   IF #Signal_AI.Value < #Signal_AI.Scal_Min_Eu THEN      //Ïðè âûõîäå çíà÷åíèÿ ñèãíàëà èç çàäàííîãî äèàïàçîíà ïðèðàâíèâàåì åãî ê íèæíåìó ïðåäåëó  ýòîãî äèàïàçîíà
       #Signal_AI.Value := #Signal_AI.Scal_Min_Eu;
       #Signal_AI.Scal_Min_Under := true;                 //çàæèãàåì ôëàã  çíà÷åíèÿ ñèãíàëà íèæå íèæíåãî ïðåäåëà äèàïàçîíà ìàñøòàáèðîâàíèÿ
   ELSE
       #Signal_AI.Scal_Min_Under := false;
   END_IF;

   //------------------------------------------------------------------------
   //---------Áëîê ïðîâåðêè ïðåâûøåíèÿ óñòàâêè ïî âåðõíåìó àâàðèéíîìó ïðåäåëó
   //------------------------------------------------------------------------
   IF #Signal_AI.HH_Alarm THEN    // Åñëè åñòü àâàðèÿ òî äëÿ îáåñïå÷åíèÿ ãèñòåðåçèñà 
       // Ðàçðåøåíèå íà ñòàðò òàéìåðà åñëè ïðîâåðêà ðàçðåøåíà è çíà÷åíèå ïðåâûøàåò óñòàâêó
       #Temp_Start_Timer := #Signal_AI.HH_Alarm_En AND (#Signal_AI.Value > (#Signal_AI.HH_Lim - #Signal_AI.HH_DeadBand));
   ELSE
       // Ðàçðåøåíèå íà ñòàðò òàéìåðà åñëè ïðîâåðêà ðàçðåøåíà è çíà÷åíèå ïðåâûøàåò óñòàâêó
       #Temp_Start_Timer := #Signal_AI.HH_Alarm_En AND (#Signal_AI.Value > (#Signal_AI.HH_Lim + #Signal_AI.HH_DeadBand));
   END_IF;

   #HH_Timer(IN := #Temp_Start_Timer // IN: BOOL
             ,
             PT := #Signal_AI.HH_Delay // IN: TIME
   );

   //åñëè  âðåìÿ çàäåðæêè èñòåêëî òî çàæèãàåì ôëàã àâàðèè , èíà÷å ãàñèì åãî
   IF #HH_Timer.Q THEN
       #Signal_AI.HH_Alarm := true;
       #Signal_AI.State := #Signal_AI.State OR #UEL;
   ELSE
       #Signal_AI.HH_Alarm := false;
       #Signal_AI.State := #Signal_AI.State AND (NOT (#UEL));
   END_IF;

   //------------------------------------------------------------------------
   //Áëîê ïðîâåðêè ïðåâûøåíèÿ óñòàâêè ïî âåðõíåìó ïðåäóïðåäèòåëüíîìó ïðåäåëó
   //------------------------------------------------------------------------
   IF #Signal_AI.H_Alarm THEN    // Åñëè åñòü àâàðèÿ òî äëÿ îáåñïå÷åíèÿ ãèñòåðåçèñà 
       // Ðàçðåøåíèå íà ñòàðò òàéìåðà åñëè ïðîâåðêà ðàçðåøåíà è çíà÷åíèå ïðåâûøàåò óñòàâêó
       #Temp_Start_Timer := #Signal_AI.H_Alarm_En AND (#Signal_AI.Value > (#Signal_AI.H_Lim - #Signal_AI.H_DeadBand));
   ELSE
       // Ðàçðåøåíèå íà ñòàðò òàéìåðà åñëè ïðîâåðêà ðàçðåøåíà è çíà÷åíèå ïðåâûøàåò óñòàâêó
       #Temp_Start_Timer := #Signal_AI.H_Alarm_En AND (#Signal_AI.Value > (#Signal_AI.H_Lim + #Signal_AI.H_DeadBand));
   END_IF;

   #H_Timer(IN := #Temp_Start_Timer // IN: BOOL
            ,
            PT := #Signal_AI.H_Delay // IN: TIME
   );

   //åñëè  âðåìÿ çàäåðæêè èñòåêëî òî çàæèãàåì ôëàã àâàðèè , èíà÷å ãàñèì åãî
   IF #H_Timer.Q THEN
       #Signal_AI.H_Alarm := true;
       #Signal_AI.State := #Signal_AI.State OR #UWL;
   ELSE
       #Signal_AI.H_Alarm := false;
       #Signal_AI.State := #Signal_AI.State AND (NOT (#UWL));
   END_IF;

   //------------------------------------------------------------------------
   //--Áëîê ïðîâåðêè ïðåâûøåíèÿ óñòàâêè ïî íèæíåìó ïðåäóïðåäèòåëüíîìó ïðåäåëó
   //------------------------------------------------------------------------
   IF #Signal_AI.L_Alarm THEN    // Åñëè åñòü àâàðèÿ òî äëÿ îáåñïå÷åíèÿ ãèñòåðåçèñà 
       #Temp_Start_Timer := #Signal_AI.L_Alarm_En AND (#Signal_AI.Value < (#Signal_AI.L_Lim + #Signal_AI.L_DeadBand));   // Ðàçðåøåíèå íà ñòàðò òàéìåðà åñëè ïðîâåðêà ðàçðåøåíà è çíà÷åíèå ïðåâûøàåò óñòàâêó
   ELSE
       #Temp_Start_Timer := #Signal_AI.L_Alarm_En AND (#Signal_AI.Value < (#Signal_AI.L_Lim - #Signal_AI.L_DeadBand));   // Ðàçðåøåíèå íà ñòàðò òàéìåðà åñëè ïðîâåðêà ðàçðåøåíà è çíà÷åíèå ïðåâûøàåò óñòàâêó
   END_IF;

   #L_Timer(IN := #Temp_Start_Timer // IN: BOOL
            ,
            PT := #Signal_AI.L_Delay // IN: TIME
   );

   //åñëè  âðåìÿ çàäåðæêè èñòåêëî òî çàæèãàåì ôëàã àâàðèè , èíà÷å ãàñèì åãî
   IF #L_Timer.Q THEN
       #Signal_AI.L_Alarm := true;
       #Signal_AI.State := #Signal_AI.State OR #DWL;
   ELSE
       #Signal_AI.L_Alarm := false;
       #Signal_AI.State := #Signal_AI.State AND (NOT (#DWL));
   END_IF;

   //------------------------------------------------------------------------
   //-------Áëîê ïðîâåðêè ïðåâûøåíèÿ óñòàâêè ïî íèæíåìó àâàðèéíîìó ïðåäåëó---
   //------------------------------------------------------------------------
   IF #Signal_AI.LL_Alarm THEN    // Åñëè åñòü àâàðèÿ òî äëÿ îáåñïå÷åíèÿ ãèñòåðåçèñà 
       #Temp_Start_Timer := #Signal_AI.LL_Alarm_En AND (#Signal_AI.Value < (#Signal_AI.LL_Lim + #Signal_AI.LL_DeadBand));   // Ðàçðåøåíèå íà ñòàðò òàéìåðà åñëè ïðîâåðêà ðàçðåøåíà è çíà÷åíèå ïðåâûøàåò óñòàâêó
   ELSE
       #Temp_Start_Timer := #Signal_AI.LL_Alarm_En AND (#Signal_AI.Value < (#Signal_AI.LL_Lim - #Signal_AI.LL_DeadBand));   // Ðàçðåøåíèå íà ñòàðò òàéìåðà åñëè ïðîâåðêà ðàçðåøåíà è çíà÷åíèå ïðåâûøàåò óñòàâêó
   END_IF;

   #LL_Timer(IN := #Temp_Start_Timer // IN: BOOL
             ,
             PT := #Signal_AI.LL_Delay // IN: TIME
   );

   //åñëè  âðåìÿ çàäåðæêè èñòåêëî òî çàæèãàåì ôëàã àâàðèè , èíà÷å ãàñèì åãî
   IF #LL_Timer.Q THEN
       #Signal_AI.LL_Alarm := true;
       #Signal_AI.State := #Signal_AI.State OR #DEL;
   ELSE
       #Signal_AI.LL_Alarm := false;
       #Signal_AI.State := #Signal_AI.State AND (NOT (#DEL));
   END_IF;

   //Определяем состояние маскирования
   IF (#Signal_AI.HH_Alarm_En AND #Signal_AI.H_Alarm_En AND #Signal_AI.L_Alarm_En AND #Signal_AI.LL_Alarm_En) THEN
       #Signal_AI.State := #Signal_AI.State AND (NOT (#MSK));// OR #MSK;
   ELSE
       #Signal_AI.State := #Signal_AI.State OR #MSK;// AND (NOT (#MSK));
   END_IF;


   //------------------------------------------------------------------------
   //------Áëîê ïðîâåðêè íà êîðîòêîå çàìûêàíèå è îáðûâ-----------------------
   //------------------------------------------------------------------------
   IF (NOT #Signal_AI.Sim_En) THEN
       // Ïðîâåðêà íà êîðîòêîå çàìûêàíèå.
       #Signal_AI.Short_Circuit := (#Signal_AI.Acp >= #ACP_sc);

       // Ïðîâåðêà íà îáðûâ.
       IF #Signal_AI.VoltageInputType AND (#Signal_AI.Resistance > 0) THEN
           // âõîä íàïðÿæåíèÿ ñ ïðåîáðàçîâàíèåì â òîêîâûé
           IF #Signal_AI.Scale_0_20mA THEN
               #Signal_AI.Break := (#Signal_AI.Circuit <= #Curr0_20_br);
           ELSE
               #Signal_AI.Break := (#Signal_AI.Circuit <= #Curr4_20_br);
           END_IF;
       ELSE
           // òîêîâûé âõîä
           IF (#Signal_AI.Scale_0_20mA AND #Signal_AI.Input_4mA_on_0_20mA) THEN
               #Signal_AI.Break := (#Signal_AI.Circuit <= #Curr4_20_br);
           ELSE
               #Signal_AI.Break := (#Signal_AI.Acp <= #ACP_br);
           END_IF;
       END_IF;


       //  Ïðè îáðûâå èëè êîðîòêîì çàìûêàíèè  ãàñèì ôëàãè ñðàáàòûâàíèÿ óñòàâîê
       IF (#Signal_AI.Short_Circuit OR #Signal_AI.Break) THEN
           #Signal_AI.HH_Alarm := false;
           #Signal_AI.H_Alarm := false;
           #Signal_AI.L_Alarm := false;
           #Signal_AI.LL_Alarm := false;
           #Signal_AI.Chan_Fail := true;
           #Signal_AI.State := #Signal_AI.State OR #PNC;
       ELSE
           #Signal_AI.Chan_Fail := false;
           #Signal_AI.State := #Signal_AI.State AND (NOT (#PNC));
       END_IF;

   ELSE
       #Signal_AI.Short_Circuit := false;
       #Signal_AI.Break := false;
       #Signal_AI.Chan_Fail := false;
   END_IF;

   // Режим маскирования (или тестирования ?) - ХЗ. сделал как-будто это одно и то же
   IF (#Signal_AI.Mask_mode) THEN
       #Signal_AI.HH_Alarm_Logic := false;
       #Signal_AI.H_Alarm_Logic := false;
       #Signal_AI.L_Alarm_Logic := false;
       #Signal_AI.LL_Alarm_Logic := false;
       #Signal_AI.Chan_Fail_Logic := false;
       #Signal_AI.Test_mode := true;
   ELSE
       #Signal_AI.HH_Alarm_Logic := #Signal_AI.HH_Alarm;
       #Signal_AI.H_Alarm_Logic := #Signal_AI.H_Alarm;
       #Signal_AI.L_Alarm_Logic := #Signal_AI.L_Alarm;
       #Signal_AI.LL_Alarm_Logic := #Signal_AI.LL_Alarm;
       #Signal_AI.Chan_Fail_Logic := #Signal_AI.Chan_Fail;
       #Signal_AI.Test_mode := false;
   END_IF;

   // Квитирование аварий по аналоговым параметрам (моргание на HMI)
   IF ((#Signal_AI.HH_Alarm AND NOT #Signal_AI.Ack_HH) OR (#Signal_AI.LL_Alarm AND NOT #Signal_AI.Ack_LL)) THEN
       #Signal_AI.Ack_Alarm := 1;
   ELSIF ((#Signal_AI.HH_Alarm AND #Signal_AI.Ack_HH) OR (#Signal_AI.LL_Alarm AND #Signal_AI.Ack_LL)) THEN
       #Signal_AI.Ack_Alarm := 2;
   ELSIF (NOT #Signal_AI.HH_Alarm AND NOT #Signal_AI.LL_Alarm) THEN
       #Signal_AI.Ack_Alarm := 0;
       #Signal_AI.Ack_HH := false;
       #Signal_AI.Ack_LL := false;
   END_IF;

   IF ((#Signal_AI.H_Alarm AND NOT #Signal_AI.Ack_H) OR (#Signal_AI.L_Alarm AND NOT #Signal_AI.Ack_L)) THEN
       #Signal_AI.Ack_Warning := 1;
   ELSIF ((#Signal_AI.H_Alarm AND #Signal_AI.Ack_H) OR (#Signal_AI.L_Alarm AND #Signal_AI.Ack_L)) THEN
       #Signal_AI.Ack_Warning := 2;
   ELSIF (NOT #Signal_AI.H_Alarm AND NOT #Signal_AI.L_Alarm) THEN
       #Signal_AI.Ack_Warning := 0;
       #Signal_AI.Ack_H := false;
       #Signal_AI.Ack_L := false;
   END_IF;

   // Закраска прямоугольников на HMI
   IF (#Signal_AI.Mask_mode) THEN
       #Signal_AI.State_color := 3;
   ELSIF (#Signal_AI.Chan_Fail) THEN
       #Signal_AI.State_color := 4;
   ELSIF (#Signal_AI.HH_Alarm OR #Signal_AI.LL_Alarm) THEN
       #Signal_AI.State_color := 2;
   ELSIF (#Signal_AI.H_Alarm OR #Signal_AI.L_Alarm) THEN
       #Signal_AI.State_color := 1;
   ELSE
       #Signal_AI.State_color := 0;
   END_IF;
END_FUNCTION_BLOCK

FUNCTION_BLOCK "Scan_Dev"   // FB2, SCL
{ S7_Optimized_Access := 'FALSE' }
NAME : Scan_Dev
VERSION : 1.2
   VAR_INPUT
      IN_State_OnOff : Bool;   // On/Off state of device (Common state input)
      IN_State_On : Bool;   // On state of device (Separate state inputs)
      IN_State_Off : Bool;   // Off state of device (Separate state inputs)
      IN_ModeLocal : Bool;   // 0 - local control, 1 - remote control (device switch)
   END_VAR
   VAR_OUTPUT
      OUT_CMD_ON : Bool;   // Switch On command
      OUT_CMD_OFF : Bool;   // Switch Off command
   END_VAR
   VAR
      Device : Struct
         Cmd_On : Byte;   // Switch On commands : 0-None, 1-local, 2-remote auto, 4-remote manual(SCADA), 8-remote manual(OP)
         Cmd_Off : Byte;   // Switch Off commands: 0-None, 1-local, 2-remote auto, 4-remote manual(SCADA), 8-remote manual(OP)
         Mode : Byte := 4;   // Operate mode: 1-local, 2-remote auto, 4-remote manual(SCADA), 8-remote manual(OP), 16-Repair
         Fail : Byte;   // Fail (0-None, 128-common failure)
         State : Byte;   // Device state (0-off,1-on, 128-undefine)
         Control_Lock : Byte;   // Outer protection lock of device (0 - no protection, can work)
         Cfg_Time_OnOff : Time := T#5S;   // switch time (second)
         Cfg_OutPulseLen : Time := T#3S;   // Command pulse delay (second)
         RunTime : Real := 0.0;   // Worktime from last start (second)
         RunTime_Total : Real := 0.0;   // Total Worktime from last reset (second)
         RunTime_LastScan : Date_And_Time;   // Intermediate worktime (DTL)
         Sim_State : Byte;   // Device simulating state (0-off,1-on, 128-undefine)
         Sim_En : Bool;   // Simulate enable
         On_Flag : Bool := FALSE;   // On command accepted
         Off_Flag : Bool := FALSE;   // Off command accapted
         On_output : Bool := 0;   // On output state
         Off_output : Bool := 0;   // Off output state
         Cfg_OutputLevelCmd : Bool := FALSE;   // Output command type: false-pulse, true-level
         Cfg_TwoStateInputs : Bool := FALSE;   // Number of device state inputs: false-one common input, true-two separate inputs
         Cfg_CalculateRuntime : Bool := TRUE;   // true - calculate worktime
         Cfg_IgnoreStateInputs : Bool := FALSE;   // true - execute commands in any device state
         Cmd_Reset_Error : Byte;
         Reset_Error_Flag : Bool;
         Reset_Error_Output : Bool;
         auto : Bool;
      END_STRUCT;
      Device_Timer : TON_TIME;
      Cfg_Time_OnOff : DInt;
      Cfg_Time_OnOff_1 : DInt;
   END_VAR
   VAR_TEMP
      Temp_Start_Timer : Bool;
      Temp_Timer_Counting : Bool;
      Temp_Reset_Timer : Bool;
      Temp_Timer_State : Bool;
      Temp_Int : Int;
      Temp_CurTime : Time;
      Temp_Time : Time;
      temp_dint : DInt;
      CurrentTime : Date_And_Time;
      curr_TOD : Time_Of_Day;
      BDR_flag_ON : Bool;
      BDR_flag_OFF : Bool;
   END_VAR
BEGIN

   // 0)При инициализации (в OB100) необходимо сбрасывать Device.RunTime_LastScan в DTL#1970-1-1-0:0:0.0, иначе будет врать наработка 
   // 1)Каждому устройству необходимо выставить время включения-отключения  устройства (Cfg_Time_OnOf)
   // 2)Каждому устройству необходимо выставить тип управления (Cfg_TypeControl), 0-импульное, 1-постоянное 
   // 3)Каждому устройству необходимо выставить время длительности выходного импульса (Cfg_Time_Imp), если используется импульсный тип управления.                                                                     *//
   // 4)Каждому устройству выставить число входных сигналов состояния устройства Cfg_TwoStateInputs (True - 2 параметра, False - 1 параметр)


   // Обработки режима симуляции и определения состояния устройства

   //Если режим симуляции включен то заменяем ходные значение на значение для симуляции   
   IF #Device.Sim_En THEN
       #Device.State := #Device.Sim_State;
   ELSE
       // Если два входа состояния устройства
       IF #Device.Cfg_TwoStateInputs THEN
           IF #IN_State_Off THEN
               #Device.State := 2#00000000;                 // Состояние, Устройство выключено
           END_IF;
           IF #IN_State_On THEN
               #Device.State := 2#00000001;                 // Состояние, Устройство включено
           END_IF;
           IF NOT (#IN_State_Off XOR #IN_State_On) THEN       // Концевики оба =1 или =0 то
               #Device.State := 2#10000000;                 // Состояние, устройство неопределено
               #Device.Fail := #Device.Fail OR 2#00000100;   // Код аварии (4) - неопределенное значение концевиков
           END_IF;
       ELSE
           // Если один вход состояния устройства
           IF #IN_State_OnOff THEN
               #Device.State := 2#00000001;                 // Состояние, Устройство включено
           ELSE
               #Device.State := 2#00000000;                 // Состояние, Устройство выключено
           END_IF;
       END_IF;

       // Если состояние от переключателя - местн. режим то устанавливаем его иначе скидываем
       IF #IN_ModeLocal THEN
           #Device.Mode := #Device.Mode OR 2#00000001;
       ELSE
           #Device.Mode := #Device.Mode AND 2#11111110;
       END_IF;
   END_IF;



   // Обработка команд в соответствии с выбранным режимом управления и наличия аварии

   #Temp_Reset_Timer := false;

   // Если нет внешней аварии для блокировки управления устройством то можно включать устройство
   IF (#Device.Control_Lock = 0) THEN

       // Если есть команда на включение и она соответствует режиму управления
       IF (#Device.Mode AND #Device.Cmd_On) <> 0 THEN
           // Если состояние устройство не включено или мы игнорируем состояние устройства
           IF ((#Device.State AND 2#00000001) = 0) OR (#Device.Cfg_IgnoreStateInputs) THEN
               // Если флаг по команде управления на включение не зажжен, то обработаем команду однократно
               IF NOT #Device.On_Flag THEN

                   #Device.Fail := 0;                    // Сброс внутренней аварии

                   #Device.On_output := TRUE;          // Однократно по полож. фронту зажигаем внутреннюю команду на включение устройства
                   #Device.On_Flag := TRUE;          // Однократно по полож. фронту зажигаем флаг сигнализации что команда прошла

                   #Device.Off_Flag := FALSE;        // Однократно по полож. фронту сбрасываем флаг сигнализации что команда прошла
                   #Device.Off_output := FALSE;        // Однократно по полож. фронту сбрасываем внутреннюю команду на выключение

                   #Temp_Reset_Timer := TRUE;            // Однократно по полож. фронту команды сбрасываем таймер работы устройства  

               END_IF;
           END_IF;
       ELSE
           #Device.On_Flag := FALSE;                // Однократно по полож. фронту сбрасываем флаг сигнализации что команда прошла
       END_IF;

       // Если есть команда на выключение и она соответствует режиму управления
       IF (#Device.Mode AND #Device.Cmd_Off) <> 0 THEN
           // Если состояние устройство не выключено или мы игнорируем состояние устройства
           IF ((#Device.State AND 2#00000001) <> 0) OR (#Device.Cfg_IgnoreStateInputs) THEN
               // Если флаг по команде управления на выключение не зажжен, то обработаем команду однократно                     
               IF NOT #Device.Off_Flag THEN

                   #Device.Fail := 0;                    // Сброс внутренней аварии

                   #Device.On_output := false;         // Однократно по полож. фронту сбрасываем внутреннюю команду на включение устройства
                   #Device.On_Flag := FALSE;         // Однократно по полож. фронту сбрасываем флаг сигнализации что команда прошла

                   #Device.Off_Flag := TRUE;         // Однократно по полож. фронту зажигаем флаг сигнализации что команда прошла
                   #Device.Off_output := TRUE;         // Однократно по полож. фронту зажигаем внутреннюю команду на выключение

                   #Temp_Reset_Timer := TRUE;            // Однократно по полож. фронту команды сбрасываем таймер работы устройства

               END_IF;
           END_IF;
       ELSE
           #Device.Off_Flag := FALSE;                // Однократно по полож. фронту сбрасываем флаг сигнализации что команда прошла
       END_IF;

   END_IF;     //  IF ( Device.Control_Lock = 0) THEN


   IF (#Device.Mode AND #Device.Cmd_Reset_Error) <> 0 THEN
       // Если флаг по команде управления на сброс аварии не зажжен, то обработаем команду однократно                     
       IF NOT #Device.Reset_Error_Flag THEN

           #Device.Reset_Error_Output := TRUE;   // Однократно по полож. фронту зажигаем внутреннюю команду на сброс аварии устройства
           #Device.Reset_Error_Flag := TRUE;     // Однократно по полож. фронту зажигаем флаг сигнализации что команда прошла

           #Temp_Reset_Timer := TRUE;            // Однократно по полож. фронту команды сбрасываем таймер работы устройства
           #Device.Fail := 0;
           #Device.Off_Flag := false;
           #Device.On_Flag := false;
       END_IF;

   END_IF;
   #Device.Reset_Error_Flag := FALSE;    // Однократно по полож. фронту сбрасываем флаг сигнализации что команда прошла

   // команды не должны висеть - сбрасываем всё, что есть
   #Device.Cmd_On := 0;
   #Device.Cmd_Off := 0;
   #Device.Cmd_Reset_Error := 0;






   // Инициализация таймера


   // признак того, что таймер запущен, но ещё не досчитал до конца
   #Temp_Timer_Counting := (NOT #Device_Timer.Q) AND (#Device_Timer.ET > T#0ms);

   // Разрешение на старт таймера если есть команды на включение/выключение
   #Temp_Start_Timer := (NOT #Temp_Reset_Timer) AND (#Device.On_output OR #Device.Off_output);
   #Device_Timer(IN := #Temp_Start_Timer      // IN: BOOL
                 ,
                 PT := #Device.Cfg_Time_OnOff // IN: TIME
                 ,
                 ET => #Temp_CurTime);    // OUT: TIME

   // Снимаем флаг сброса таймера
   IF #Temp_Reset_Timer THEN
       #Temp_Reset_Timer := FALSE;
   END_IF;

   (*IF #Device.Fail = 2#10000001 AND #BDR_flag_ON THEN
     #OUT_CMD_OFF    := 0;
     #BDR_flag_ON  := false;
   END_IF;

   IF #Device.Fail = 2#10000011 AND #BDR_flag_OFF THEN
     #OUT_CMD_ON    := 0;
     #BDR_flag_OFF  := false;
    END_IF;*)
    //Формирование выходов при постоянном и импульсном типе управления

    // Если тип управления постоянный сигнал
    IF #Device.Cfg_OutputLevelCmd THEN
        #OUT_CMD_ON := #Device.On_output;
        #OUT_CMD_OFF := #Device.Off_output;
    ELSE
        // Если тип управления импульсный сигнал                                                          
        // Формируем импульс длительностью Cfg_OutPulseLen, но не дольше работы таймера
        IF ((#Temp_CurTime <= #Device.Cfg_OutPulseLen) AND #Temp_Timer_Counting) THEN
            #OUT_CMD_ON := #Device.On_output;
            #OUT_CMD_OFF := #Device.Off_output;
        ELSE
            #OUT_CMD_ON := 0;
            #OUT_CMD_OFF := 0;
        END_IF;


    END_IF;


    // Проверка отработки команд

    //если  время на отработку команды вышло и устройство не включилось или не выключилось то зажигаем аварию
    IF (#Device_Timer.Q) THEN
        // есть команда на включение
        IF #Device.On_output THEN
            IF ((#Device.State AND 2#00000001) = 0) THEN    // устройство не включилось
                #Device.Fail := #Device.Fail OR 2#00000001;   // Код аварии (1) - истекло время отработки команды

                //#Device.Cmd_Off := 16#04;//условие необходимое для вклчючение насоса бдр (modbus rtu)

            END_IF;
            #Device.On_output := 0;

        END_IF;
        // есть команда на выключение
        IF #Device.Off_output THEN
            IF (#Device.State AND 2#00000001) <> 0 THEN      // устройство не выключилось
                #Device.Fail := #Device.Fail OR 2#00000011;   // Код аварии (3) - истекло время отработки команды  

                // #Device.Cmd_On := 16#04;//условие необходимое для вклчючение насоса бдр (modbus rtu)
            END_IF;
            #Device.Off_output := 0;


        END_IF;
    END_IF;


    (*
    // Наработка устройства

    // Считываем текущее время контроллера
    #Temp_Int := RD_LOC_T(#CurrentTime);

    // считаем наработку только когда уже инициализвано предыдущее время
    IF (#Device.RunTime_LastScan > DTL#1970-1-1-0:0:0.0) THEN
        // если следует считать наработку и устройство включено
        IF (#Device.Cfg_CalculateRuntime AND ((#Device.State AND 2#00000001) = 1)) THEN
            #temp_dint := T_DIFF(IN1 := #CurrentTime, IN2 := #Device.RunTime_LastScan);
            #Device.RunTime := #Device.RunTime + DINT_TO_REAL(#temp_dint) * 0.001;
            #Device.RunTime_Total := #Device.RunTime_Total + DINT_TO_REAL(#temp_dint) * 0.001;
        ELSE
            #Device.RunTime := 0.0;         // Сбрасываем время наработки с последнего включения  
        END_IF;
    END_IF;

    #Device.RunTime_LastScan := #CurrentTime;

    //------------------------------------------------------------------------------------------//

    IF #Device.Fail <> 0 THEN             // Если есть какая нить авария то зажигаем общую аварию бит 8
        #Device.Fail := #Device.Fail OR 2#10000000;
    END_IF;

    #Cfg_Time_OnOff_1 := TIME_TO_DINT(#Device.Cfg_Time_OnOff);
    IF #Cfg_Time_OnOff_1 <> #Cfg_Time_OnOff * 1000 THEN
        #Device.Cfg_Time_OnOff := #Cfg_Time_OnOff * 1000;
    END_IF;
    *)
END_FUNCTION_BLOCK

FUNCTION_BLOCK "Scan_DI08"   // FB3, SCL
TITLE = '8-bit DI module scan'
{ S7_Optimized_Access := 'TRUE' }
NAME : ScanDI08
VERSION : 1.2
   VAR_INPUT
      In : Byte;
   END_VAR
   VAR
      Slot : Struct
         Input_En : Byte;   // enable input mask
         Filter_En : Byte;   // filter mask
         Invert_En : Byte;   // invert mask
         Sim_En : Byte;   // simulate enable mask
         Sim_Value : Byte;   // simulate value
         Input : Byte;   // In after inverting
         Value : Byte;   // Result after enable and filtering
         Value_Last_Scan : Byte;   // intermediate value
         Pins : Array[0..7] of Bool;   // hardware pins (accordance byte order)
      END_STRUCT;
   END_VAR
   VAR_TEMP
      Temp : Byte;
      Temp_In : Byte;
      i : Int;
   END_VAR
BEGIN



   #Temp_In := #In;
   #Slot.Input := #Temp_In XOR #Slot.Invert_En;         // Èíâåðòèðîâàíèå ñèãíàëîâ 
   #Temp_In := #Slot.Input AND #Slot.Input_En;      // Ïðîõîäÿò  òîëüêî ðàçðåøåííûå ñèíàëû     
   #Temp := #Slot.Value_Last_Scan XOR #Temp_In;   // Âûäåëåíèå áèòîâ èçìåíèâøèõñÿ çà ïåðèîä òàéìàóòà
   #Temp := #Temp AND #Slot.Filter_En;            // Ïðîâåðÿåì íàëè÷èå ðàçðåøåíèÿ íà ôèëüòðîâàíèå îò äðåáåçãà
   #Slot.Value := #Slot.Value AND #Temp;                // Ñîõðàíÿåì áèòû êîòîðûå íå äîëæíû èçìåíèòñÿ è îáíóëÿåì âñå îñòàëüíûå
   #Temp := NOT #Temp;                           // Èíâåðòèðóåì
   #Temp := #Temp AND #Temp_In;                  // Èçìåíèâøèåñÿ áèòû îáíóëÿåìè à íå èçìåíèâøèåñÿ ñ ïîñëåäíåãî ñêàíà áèòû çàïîìèíàåì 
   #Slot.Value := #Slot.Value OR #Temp;                 // Ôîðìèðóåì âûõîä 
   #Slot.Value_Last_Scan := #Temp_In;                   // Çàïîìèíàåì òåêóùåå çíà÷åíèå êàê çíà÷åíèå ïîñëåäíåãî ñêàíà

   // Ïðè âêëþ÷åííîé ñèìóëÿöèè çàìåíÿåì èñõîäíîå çíà÷åíèå íà Sim_Value
   #Slot.Value := (#Slot.Sim_En AND #Slot.Sim_Value) OR ((NOT #Slot.Sim_En) AND #Slot.Value);

   FOR #i := 0 TO 7 DO
       #Slot.Pins[#i] := "GetBitByte"(Data := #Slot.Value,
                                      pos := #i);
   END_FOR;
END_FUNCTION_BLOCK

FUNCTION_BLOCK "Put_DO08"   // FB4, SCL
TITLE = 'Puts 8-bit DO module data to Q-output'
{ S7_Optimized_Access := 'TRUE' }
NAME : PutDO08
VERSION : 1.0
   VAR_OUTPUT
      Out : Byte;
   END_VAR
   VAR
      Slot : "dt_DO";
   END_VAR
   VAR_TEMP
      Temp : Byte;
      i : Int;
   END_VAR
BEGIN


   IF #Slot.UsePinsAsInput THEN
       FOR #i := 0 TO 7 DO
           "SetBitByte"(pos := #i,
                        value := #Slot.Pins[#i],
                        Data := #Slot.Data_to_out);
       END_FOR;
   END_IF;

   #Temp := #Slot.Data_to_out XOR #Slot.Invert_En; // Èíâåðòèðîâàíèå ñèãíàëîâ  
   #Slot.Value := #Temp AND #Slot.Output_En;           // Ïðîõîäÿò  òîëüêî ðàçðåøåííûå ñèíàëû 

   // Ïðè âêëþ÷åííîé ñèìóëÿöèè çàìåíÿåì èñõîäíîå çíà÷åíèå íà Sim_Value
   #Out := (#Slot.Sim_En AND #Slot.Sim_Value) OR ((NOT #Slot.Sim_En) AND #Slot.Value);
END_FUNCTION_BLOCK

// folder: Helpers

FUNCTION "CopyWord" : Void   // FC1, SCL
{ S7_Optimized_Access := 'FALSE' }
VERSION : 0.1
   VAR_INPUT
      NDBsrc : Int;   // Номер DB-источника данных
      NDBdest : Int;   // Номер DB-приёмника данных
      offset_src : Int;   // Смещение от начала DB-источника, в байтах
      offset_dest : Int;   // Смещение от начала DB-приёмника, в байтах
      "counter" : Int;   // Число копируемых с переворотом WORD-ов
   END_VAR
   VAR_TEMP
      i : Int;
      peek1 : Word;
   END_VAR
BEGIN

   FOR #i := 0 TO (#counter - 1) DO
       #peek1 := PEEK_WORD(area := 16#84,
                           dbNumber := #NDBsrc,
                           byteOffset := #offset_src + (#i * 2));
       POKE(area := 16#84,
            dbNumber := #NDBdest,
            byteOffset := #offset_dest + (#i * 2),
            value := #peek1);
   END_FOR;
END_FUNCTION

FUNCTION "GetBitByte" : Bool   // FC2, SCL
{ S7_Optimized_Access := 'TRUE' }
VERSION : 0.1
   VAR_INPUT
      Data : Byte;
      pos : Int;
   END_VAR
   VAR_TEMP
      mask : Byte;
      temp : Byte;
   END_VAR
BEGIN
   #mask := 1;
   IF #pos < 8 THEN
       #mask := SHL(IN := #mask, N := #pos);
       #temp := #Data AND #mask;
       #GetBitByte := (#temp > 0);
   ELSE
       #GetBitByte := 0;
   END_IF;
END_FUNCTION

FUNCTION "GetBitWord" : Bool   // FC3, SCL
{ S7_Optimized_Access := 'TRUE' }
VERSION : 0.1
   VAR_INPUT
      Data : Word;
      pos : Int;
   END_VAR
   VAR_TEMP
      mask : Word;
      temp : Word;
   END_VAR
BEGIN
   #mask := 1;
   IF #pos < 16 THEN
       #mask := SHL(IN := #mask, N := #pos);
       #temp := #Data AND #mask;
       #GetBitWord := (#temp > 0);
   ELSE
       #GetBitWord := 0;
   END_IF;
END_FUNCTION

FUNCTION "SwapWord" : Void   // FC4, SCL
{ S7_Optimized_Access := 'TRUE' }
VERSION : 0.1
   VAR_INPUT
      NDB : Int;   // Номер DB-источника данных
      offset : Int;   // Смещение от начала DB, в байтах
      "counter" : Int;   // Число переворачиваемых WORD-ов
   END_VAR
   VAR_TEMP
      peek1 : Byte;
      peek2 : Byte;
      i : Int;
   END_VAR
BEGIN

   FOR #i := #offset TO #offset + (#counter - 1) * 2 BY 2 DO
       #peek1 := PEEK(area := 16#84,
                      dbNumber := #NDB,
                      byteOffset := #i);
       #peek2 := PEEK(area := 16#84,
                      dbNumber := #NDB,
                      byteOffset := #i + 1);
       POKE(area := 16#84,
            dbNumber := #NDB,
            byteOffset := #i + 1,
            value := #peek1);
       POKE(area := 16#84,
            dbNumber := #NDB,
            byteOffset := #i,
            value := #peek2);
   END_FOR;
END_FUNCTION

FUNCTION "Swap_float" : Void   // FC5, SCL
{ S7_Optimized_Access := 'TRUE' }
VERSION : 0.1
   VAR_INPUT
      offset : Int;
      "counter" : Int;
      NDB : Int;
   END_VAR
   VAR_TEMP
      i : Int;
      peek1 : Word;
      peek2 : Word;
   END_VAR
BEGIN
   FOR #i := #offset TO #offset + (#counter - 1) * 4 BY 4 DO
       #peek1 := PEEK_WORD(area := 16#84,
                           dbNumber := #NDB,
                           byteOffset := #i);
       #peek2 := PEEK_WORD(area := 16#84,
                           dbNumber := #NDB,
                           byteOffset := #i + 2);
       POKE(area := 16#84,
            dbNumber := #NDB,
            byteOffset := #i + 2,
            value := #peek1);
       POKE(area := 16#84,
            dbNumber := #NDB,
            byteOffset := #i,
            value := #peek2);
   END_FOR;
END_FUNCTION

FUNCTION "SetBitWord" : Void   // FC6, SCL
{ S7_Optimized_Access := 'TRUE' }
VERSION : 0.1
   VAR_INPUT
      pos : Int;
      value : Bool;
   END_VAR
   VAR_IN_OUT
      Data : Word;
   END_VAR
   VAR_TEMP
      mask : Word;
      v : Word;
   END_VAR
BEGIN
   IF #pos < 16 THEN
       #mask := 1;
       #mask := SHL(IN := #mask, N := #pos);
       IF #value THEN
           #Data := #Data OR #mask;
       ELSE
           #Data := #Data AND (NOT #mask);
       END_IF;
   END_IF;
END_FUNCTION

FUNCTION "SetBitByte" : Void   // FC7, SCL
{ S7_Optimized_Access := 'TRUE' }
VERSION : 0.1
   VAR_INPUT
      pos : Int;
      value : Bool;
   END_VAR
   VAR_IN_OUT
      Data : Byte;
   END_VAR
   VAR_TEMP
      mask : Byte;
      v : Byte;
   END_VAR
BEGIN
   IF #pos < 8 THEN
       #mask := 1;
       #mask := SHL(IN := #mask, N := #pos);
       IF #value THEN
           #Data := #Data OR #mask;
       ELSE
           #Data := #Data AND (NOT #mask);
       END_IF;
   END_IF;
END_FUNCTION

// folder: Modbus

FUNCTION "UVP_Processing" : Void   // FC9, SCL
{ S7_Optimized_Access := 'TRUE' }
VERSION : 0.1
   VAR_TEMP
      NewState : Int;
      Cant_connect1 : Bool;
      Cant_connect2 : Bool;
      Cant_connect_with_UVP : Bool;
      Request_Finished : Bool;
      Request_Finished_with_Error : Bool;
      len : UInt;
   END_VAR
BEGIN
   // Установить IP адрес УВП
   (*IF "UVP_Data".Commands.Set_IP_UVP1 THEN
       IF NOT "UVP_States".Client.Disconnect THEN
           "UVP_States".Connect_UVP.ID := UINT_TO_WORD("UVP_Data".UVP1_Settings.Connect_ID);
           "UVP_States".Connect_UVP.RemoteAddress.ADDR[1] := UINT_TO_BYTE("UVP_Data".UVP1_Settings.IP_OCTET1);
           "UVP_States".Connect_UVP.RemoteAddress.ADDR[2] := UINT_TO_BYTE("UVP_Data".UVP1_Settings.IP_OCTET2);
           "UVP_States".Connect_UVP.RemoteAddress.ADDR[3] := UINT_TO_BYTE("UVP_Data".UVP1_Settings.IP_OCTET3);
           "UVP_States".Connect_UVP.RemoteAddress.ADDR[4] := UINT_TO_BYTE("UVP_Data".UVP1_Settings.IP_OCTET4);
           "UVP_States".Connect_UVP.RemotePort := "UVP_Data".UVP1_Settings.IP_PORT;
           "UVP_States".State := 10;
           "UVP_States".Client.Disconnect := True;
       ELSE
           "UVP_States".Client.Disconnect := False;
           "UVP_Data".Commands.Set_IP_UVP1 := False;
       END_IF;
   END_IF;*)

   #NewState := -1;

   // определение проблем с подключением
   #Request_Finished := "UVP_States".Client.Done OR "UVP_States".Client.Error OR ("UVP_States".Client.Busy AND ("UVP_States".Client.Status = 16#7002));
   // признак завершения цикла работы чтения/записи с ошибкой
   #Request_Finished_with_Error := ("UVP_States".Client.Busy AND ("UVP_States".Client.Status = 16#7002)) OR
   ("UVP_States".Client.Error AND (("UVP_States".Client.Status <> 16#7002)));

   // определение проблем со связью
   IF ("UVP_States".Client.Busy OR "UVP_States".Client.Error) THEN
       "UVP_off".TON (IN := true, PT := t#5s);
       IF "UVP_off".Q THEN
           "UVP_Data".Flags.UVP1_on := false;
           "ReqUVP" := 0;
           #NewState := "UVP_States".ReqReadOpData_nextState;
           "UVP_off".TON (IN := false, PT := t#5s);
       END_IF;
   ELSE
       "UVP_off".TON (IN := false, PT := t#5s);
   END_IF;

   IF "UVP_States".Client.Done AND (NOT "UVP_States".Client.Error) THEN
       "UVP_Data".Flags.UVP1_on := true;
   END_IF;

   CASE "UVP_States".State OF
       10..29:// State=10 - чтение оперативных данных первой линии, параметры с 3 по 23
              // State=11 - чтение накопленных данных первой линии, 4 группы по 5 параметров
              // 
              // State=13 - чтение оперативных данных второй линии, параметры с 3 по 23
              // State=14 - чтение накопленных данных второй линии, 4 группы по 5 параметров
              // 
              // State=16 - чтение оперативных данных второй линии, параметры с 3 по 23
              // State=17 - чтение накопленных данных второй линии, 4 группы по 5 параметров

           IF ("PrevState" <> "UVP_States".State) THEN
               "UVP_States".ReqReadOpData.Mode := 0;
               //ил 1
               IF "UVP_States".State = 10 THEN
                   "UVP_States".ReqReadOpData.Data_ADDR := 32001;
                   "UVP_States".ReqReadOpData.Data_LEN := 46;
                   "UVP_States".ReqReadOpData_dest_offset := 64; // смещение проверить в Дата
                   "UVP_States".ReqReadOpData_nextState := 11;
               ELSIF "UVP_States".State = 11 THEN
                   "UVP_States".ReqReadOpData.Data_ADDR := 32061;
                   "UVP_States".ReqReadOpData.Data_LEN := 40;
                   "UVP_States".ReqReadOpData_dest_offset := 156; // смещение проверить в Дата
                   "UVP_States".ReqReadOpData_nextState := 13;

                   //ил 2    
               ELSIF "UVP_States".State = 13 THEN
                   "UVP_States".ReqReadOpData.Data_ADDR := 32101;
                   "UVP_States".ReqReadOpData.Data_LEN := 46;
                   "UVP_States".ReqReadOpData_dest_offset := 236;
                   "UVP_States".ReqReadOpData_nextState := 14;
               ELSIF "UVP_States".State = 14 THEN
                   "UVP_States".ReqReadOpData.Data_ADDR := 32161;
                   "UVP_States".ReqReadOpData.Data_LEN := 40;
                   "UVP_States".ReqReadOpData_dest_offset := 328;
                   "UVP_States".ReqReadOpData_nextState := 16;

                   //ил 3    
               ELSIF "UVP_States".State = 16 THEN
                   "UVP_States".ReqReadOpData.Data_ADDR := 32201;
                   "UVP_States".ReqReadOpData.Data_LEN := 46;
                   "UVP_States".ReqReadOpData_dest_offset := 408;
                   "UVP_States".ReqReadOpData_nextState := 17;
               ELSIF "UVP_States".State = 17 THEN
                   "UVP_States".ReqReadOpData.Data_ADDR := 32261;
                   "UVP_States".ReqReadOpData.Data_LEN := 40;
                   "UVP_States".ReqReadOpData_dest_offset := 500;//
                   "UVP_States".ReqReadOpData_nextState := 30;
               END_IF;
               "ReqUVP" := 0;
               "UVP_States".ClientMode := "UVP_States".ReqReadOpData;
               "ReqUVP" := 1;

           END_IF;
           // обработка принятых данных
           IF "UVP_States".Client.Done THEN
               // перекладываем прочитаные данные в секцию UVP_Current_L1(L2), UVP_Current_L1(L2)  или UVP_Cumulative_L1(L3), смотря по запросу              
               "CopyWord"(NDBsrc := 14,
                          NDBdest := 13,
                          offset_src := 52,
                          offset_dest := "UVP_States".ReqReadOpData_dest_offset,
                          counter := UINT_TO_INT("UVP_States".ReqReadOpData.Data_LEN));
               "ReqUVP" := 0;
               // постобработка данных - перевожу Па в МПа, секундные расходы в часовые
               IF "UVP_States".State = 10 THEN
                   "UVP_Data".UVP1_Current_L1.UVP_mass_flow := "UVP_Data".UVP1_Current_L1.UVP_mass_flow * 3600.0;
                   "UVP_Data".UVP1_Current_L1.UVP_Param_m_flow := "UVP_Data".UVP1_Current_L1.UVP_Param_m_flow * 3600.0;
                   "UVP_Data".UVP1_Current_L1.UVP_Param_vol_flow_norm := "UVP_Data".UVP1_Current_L1.UVP_Param_vol_flow_norm * 3600.0;
                   "UVP_Data".UVP1_Current_L1.UVP_Param_vol_flow_work := "UVP_Data".UVP1_Current_L1.UVP_Param_vol_flow_work * 3600.0;
                   "UVP_Data".UVP1_Current_L1.UVP_vol_flow_norm := "UVP_Data".UVP1_Current_L1.UVP_vol_flow_norm * 3600.0;
                   "UVP_Data".UVP1_Current_L1.UVP_vol_flow_work := "UVP_Data".UVP1_Current_L1.UVP_vol_flow_work * 3600.0;
                   "UVP_Data".UVP1_Current_L1.UVP_Abs_press := "UVP_Data".UVP1_Current_L1.UVP_Abs_press / 1000000;
                   "UVP_Data".UVP1_Current_L1.UVP_Press := "UVP_Data".UVP1_Current_L1.UVP_Press / 1000000;
               ELSIF "UVP_States".State = 11 THEN
                   "UVP_Data".UVP1_Cumulative_L1.UVP_Mass_prev2h := "UVP_Data".UVP1_Cumulative_L1.UVP_Mass_prev2h / 1000.0;
                   "UVP_Data".UVP1_Cumulative_L1.UVP_Param_m_flow_prev2h := "UVP_Data".UVP1_Cumulative_L1.UVP_Param_m_flow_prev2h / 1000.0;
                   "UVP_Data".UVP1_Cumulative_L1.UVP_Mass_prevDay := "UVP_Data".UVP1_Cumulative_L1.UVP_Mass_prevDay / 1000.0;
                   "UVP_Data".UVP1_Cumulative_L1.UVP_Param_m_flow_prevDay := "UVP_Data".UVP1_Cumulative_L1.UVP_Param_m_flow_prevDay / 1000.0;
               ELSIF "UVP_States".State = 13 THEN
                   "UVP_Data".UVP1_Current_L2.UVP_mass_flow := "UVP_Data".UVP1_Current_L2.UVP_mass_flow * 3.6;
                   "UVP_Data".UVP1_Current_L2.UVP_Param_m_flow := "UVP_Data".UVP1_Current_L2.UVP_Param_m_flow * 3600.0;
                   "UVP_Data".UVP1_Current_L2.UVP_Param_vol_flow_norm := "UVP_Data".UVP1_Current_L2.UVP_Param_vol_flow_norm * 3600.0;
                   "UVP_Data".UVP1_Current_L2.UVP_Param_vol_flow_work := "UVP_Data".UVP1_Current_L2.UVP_Param_vol_flow_work * 3600.0;
                   "UVP_Data".UVP1_Current_L2.UVP_vol_flow_norm := "UVP_Data".UVP1_Current_L2.UVP_vol_flow_norm * 3600.0;
                   "UVP_Data".UVP1_Current_L2.UVP_vol_flow_work := "UVP_Data".UVP1_Current_L2.UVP_vol_flow_work * 3600.0;
                   "UVP_Data".UVP1_Current_L2.UVP_Abs_press := "UVP_Data".UVP1_Current_L2.UVP_Abs_press / 1000000;
                   "UVP_Data".UVP1_Current_L2.UVP_Press := "UVP_Data".UVP1_Current_L2.UVP_Press / 1000000;
               ELSIF "UVP_States".State = 14 THEN
                   "UVP_Data".UVP1_Cumulative_L2.UVP_Mass_prev2h := "UVP_Data".UVP1_Cumulative_L2.UVP_Mass_prev2h / 1000.0;
                   "UVP_Data".UVP1_Cumulative_L2.UVP_Param_m_flow_prev2h := "UVP_Data".UVP1_Cumulative_L2.UVP_Param_m_flow_prev2h / 1000.0;
                   "UVP_Data".UVP1_Cumulative_L2.UVP_Mass_prevDay := "UVP_Data".UVP1_Cumulative_L2.UVP_Mass_prevDay / 1000.0;
                   "UVP_Data".UVP1_Cumulative_L2.UVP_Param_m_flow_prevDay := "UVP_Data".UVP1_Cumulative_L2.UVP_Param_m_flow_prevDay / 1000.0;
               ELSIF "UVP_States".State = 16 THEN
                   "UVP_Data".UVP1_Current_L3.UVP_mass_flow := "UVP_Data".UVP1_Current_L3.UVP_mass_flow * 3.6;
                   "UVP_Data".UVP1_Current_L3.UVP_Param_m_flow := "UVP_Data".UVP1_Current_L3.UVP_Param_m_flow * 3600.0;
                   "UVP_Data".UVP1_Current_L3.UVP_Param_vol_flow_norm := "UVP_Data".UVP1_Current_L3.UVP_Param_vol_flow_norm * 3600.0;
                   "UVP_Data".UVP1_Current_L3.UVP_Param_vol_flow_work := "UVP_Data".UVP1_Current_L3.UVP_Param_vol_flow_work * 3600.0;
                   "UVP_Data".UVP1_Current_L3.UVP_vol_flow_norm := "UVP_Data".UVP1_Current_L3.UVP_vol_flow_norm * 3600.0;
                   "UVP_Data".UVP1_Current_L3.UVP_vol_flow_work := "UVP_Data".UVP1_Current_L3.UVP_vol_flow_work * 3600.0;
                   "UVP_Data".UVP1_Current_L3.UVP_Abs_press := "UVP_Data".UVP1_Current_L3.UVP_Abs_press / 1000000;
                   "UVP_Data".UVP1_Current_L3.UVP_Press := "UVP_Data".UVP1_Current_L3.UVP_Press / 1000000;
               ELSIF "UVP_States".State = 17 THEN
                   "UVP_Data".UVP1_Cumulative_L3.UVP_Mass_prev2h := "UVP_Data".UVP1_Cumulative_L3.UVP_Mass_prev2h / 1000.0;
                   "UVP_Data".UVP1_Cumulative_L3.UVP_Param_m_flow_prev2h := "UVP_Data".UVP1_Cumulative_L3.UVP_Param_m_flow_prev2h / 1000.0;
                   "UVP_Data".UVP1_Cumulative_L3.UVP_Mass_prevDay := "UVP_Data".UVP1_Cumulative_L3.UVP_Mass_prevDay / 1000.0;
                   "UVP_Data".UVP1_Cumulative_L3.UVP_Param_m_flow_prevDay := "UVP_Data".UVP1_Cumulative_L3.UVP_Param_m_flow_prevDay / 1000.0;
               END_IF;
               // Переходим к следующему запросу
               #NewState := "UVP_States".ReqReadOpData_nextState;

          //ELSIF #Request_Finished_with_Error THEN
               // Если не получается связаться - переходим к следующему запросу и продолжаем попытки
               //#NewState := "UVP_States".ReqReadOpData_nextState;
           ELSE
               ;
           END_IF;

           //******************** проверка команд*************************************************************************************************

           IF ("DATA".StartReadArchive = 1) THEN
               // переход к чтению архивной записи
               #NewState := 60;
               //ELSIF "UVP_Data".Commands.UVP_MR113_Read THEN         //читаем циклически
               // переход к чтению компонентного состава газа
               //    #NewState := 40;
           ELSIF "UVP_Data".Commands.UVP_MR113_Write THEN
               // переход к записи компонентного состава газа
               #NewState := 50;

           ELSE
               // нет команды
               ;
           END_IF;

       30:  //  чтение часов реального времени выбранного УВП, сразу после измеряемых параметров УВП по обоим линиям         
           IF NOT "UVP_States".Client.Busy THEN
               "UVP_States".ReqReadOpData.Mode := 0;
               "UVP_States".ReqReadOpData.Data_ADDR := 41801;
               "UVP_States".ReqReadOpData.Data_LEN := 6;
               "ReqUVP" := 0;
               "UVP_States".ClientMode := "UVP_States".ReqReadOpData;
               "ReqUVP" := 1;
               #NewState := 31;
           END_IF;

       31: // обработка принятых данных часов реального времени выбранного УВП
           // крутить их не нужно, так как в УВП они в нормальном представлении
           IF "UVP_States".Client.Done THEN
               // перекладываем прочитаные данные в секцию UVP_DateTime
               "CopyWord"(NDBsrc := 14,
                          NDBdest := 13,
                          offset_src := 52,
                          offset_dest := 924,
                          counter := 6);
               "ReqUVP" := 0;
               #NewState := 32;
           ELSIF #Request_Finished_with_Error THEN
               // Если не получается связаться - переходим к следующему запросу и продолжаем попытки
               #NewState := 32;
           ELSE
               ;
           END_IF;

       32:  //  запись нужного порядка байт в 4-х байтной переменной         
           IF NOT "UVP_States".Client.Busy THEN
               "UVP_States".ReqWriteCom.Mode := 1;
               "UVP_States".ReqWriteCom.Data_ADDR := 40101;
               "UVP_States".ReqWriteCom.Data_LEN := 1;
               "ReqUVP" := 0;
               %DB14.DBW52 := 291;                                  // это 0123h
               "UVP_States".ClientMode := "UVP_States".ReqWriteCom;
               "ReqUVP" := 1;
               #NewState := 33;
           END_IF;

       33: // ожидание завершения записи порядка байт
           IF #Request_Finished THEN
               // Возвращаемся к очередному запросу (с которого нас сняли командой)
               #NewState := 40;
               "ReqUVP" := 0;
           END_IF;


       40:  // State=40 - запуск чтения компонентного состава газа
           IF NOT "UVP_States".Client.Busy THEN
               "UVP_States".ReqReadOpData.Mode := 0;
               "UVP_States".ReqReadOpData.Data_ADDR := 41103;
               "UVP_States".ReqReadOpData.Data_LEN := 30;
               "ReqUVP" := 0;
               "UVP_States".ClientMode := "UVP_States".ReqReadOpData;
               "ReqUVP" := 1;
               #NewState := 41;
           END_IF;

       41: // State=41 - обработка принятых данных компонентного состава газа
           IF "UVP_States".Client.Done THEN
               // перекладываем прочитаные данные в секцию UVP_MR113
               "CopyWord"(NDBsrc := 14,
                          NDBdest := 13,
                          offset_src := 52,
                          offset_dest := 936,
                          counter := 30);
               "ReqUVP" := 0;
               // Возвращаемся к очередному запросу (с которого нас сняли командой)
               #NewState := 42;
               "UVP_Data".Commands.UVP_MR113_Read := False;
           ELSIF #Request_Finished_with_Error THEN
               // Если не получается связаться - переходим к следующему запросу и продолжаем попытки
               #NewState := 42;
               //"UVP_v2_Data".Commands.UVP_MR113_Read := False; // Из-за этого не читает комп. состав при загрузке контроллера
           ELSE
               ;
           END_IF;


       42:  // State=42 - запуск чтения параметров: молярная или массовая концентрация,  влажность
           IF NOT "UVP_States".Client.Busy THEN
               "UVP_States".ReqReadOpData.Mode := 0;
               "UVP_States".ReqReadOpData.Data_ADDR := 41101;
               "UVP_States".ReqReadOpData.Data_LEN := 2;
               "ReqUVP" := 0;
               "UVP_States".ClientMode := "UVP_States".ReqReadOpData;
               "ReqUVP" := 1;
               #NewState := 43;
           END_IF;

       43: // State=43 - обработка принятых параметров: молярная или массовая концентрация,  влажность
           IF "UVP_States".Client.Done THEN
               // перекладываем прочитаные данные в секцию UVP_MR113
               // крутить их не нужно, так как в УВП они в нормальном представлении
               "CopyWord"(NDBsrc := 14,
                          NDBdest := 13,
                          offset_src := 52,
                          offset_dest := 996,
                          counter := 2);
               "ReqUVP" := 0;
               // Возвращаемся к очередному запросу (с которого нас сняли командой)
               #NewState := 10;
           ELSIF #Request_Finished_with_Error THEN
               // Если не получается связаться - переходим к следующему запросу и продолжаем попытки
               #NewState := 10;
           ELSE
               ;
           END_IF;// конец            

       50:  // State=50 - запись компонентного состава газа
           IF NOT "UVP_States".Client.Busy THEN
               "UVP_States".ReqWriteCom.Mode := 1;
               "UVP_States".ReqWriteCom.Data_ADDR := 41103;
               "UVP_States".ReqWriteCom.Data_LEN := 30;
               "ReqUVP" := 0;
               "CopyWord"(NDBsrc := 57,
                          NDBdest := 33,
                          offset_src := 1740,
                          offset_dest := 86,
                          counter := 30);
               "UVP_States".ClientMode := "UVP_States".ReqWriteCom;
               "ReqUVP" := 1;
               #NewState := 52;
               "UVP_Data".Commands.UVP_MR113_Write := False;
           END_IF;

       52:  // ожидание завершения записи компонентного состава газа
           IF #Request_Finished THEN
               // Возвращаемся к очередному запросу (с которого нас сняли командой)
               #NewState := 53;
           END_IF;

       53:  // State=53 - запись параметров: молярная или массовая концентрация,  влажность
           IF NOT "UVP_States".Client.Busy THEN
               "UVP_States".ReqWriteCom.Mode := 1;
               "UVP_States".ReqWriteCom.Data_ADDR := 41101;
               "UVP_States".ReqWriteCom.Data_LEN := 2;
               "ReqUVP" := 0;
               // крутить их не нужно, так как в УВП они в нормальном представлении        
               "CopyWord"(NDBsrc := 57,
                          NDBdest := 33,
                          offset_src := 1800,
                          offset_dest := 86,
                          counter := 2);
               "UVP_States".ClientMode := "UVP_States".ReqWriteCom;
               "ReqUVP" := 1;
               #NewState := 54;
               "UVP_Data".Commands.UVP_MR113_Write := False;
           END_IF;

       54:  // ожидание завершения записи молярной или массовой концентрации,  влажности
           IF #Request_Finished THEN
               // Возвращаемся к очередному запросу (с которого нас сняли командой)
               #NewState := "UVP_States".ReqReadOpData_nextState;
           END_IF;

           //---------------------------------------------------------------------------------------------------------------------               
           //------------------------------ АРХИВЫ -------------------------------------------------------------------------------         

       60: // устанавливаем первичные настройки для первого запроса
           "UVP_States".Format := 0;
           "UVP_Data".UVP1_Archives.UVP_param := 1;
           "UVP_Data".UVP1_Archives.UVP_line := 3;  // было 3
           "UVP_Data".UVP1_Archives.UVP_day := "DATA".ArchDay;
           "UVP_Data".UVP1_Archives.UVP_month := "DATA".ArchMonth;
           "UVP_Data".UVP1_Archives.UVP_year := "DATA".ArchYear;
           "UVP_Data".UVP1_Archives.UVP_hour := 0;
           "UVP_Data".UVP1_Archives.UVP_day_end := "DATA".ArchDay;
           "UVP_Data".UVP1_Archives.UVP_month_end := "DATA".ArchMonth;
           "UVP_Data".UVP1_Archives.UVP_year_end := "DATA".ArchYear;
           "UVP_Data".UVP1_Archives.UVP_hour_end := 2;
           // очищаем данные предыдущих запросов архива
           "DATA".L1_Press_0_2h := 0.0;
           "DATA".L1_Press_2_4h := 0.0;
           "DATA".L1_Press_4_6h := 0.0;
           "DATA".L1_Press_6_8h := 0.0;
           "DATA".L1_Press_8_10h := 0.0;
           "DATA".L1_Press_10_12h := 0.0;
           "DATA".L1_Press_12_14h := 0.0;
           "DATA".L1_Press_14_16h := 0.0;
           "DATA".L1_Press_16_18h := 0.0;
           "DATA".L1_Press_18_20h := 0.0;
           "DATA".L1_Press_20_22h := 0.0;
           "DATA".L1_Press_22_24h := 0.0;
           "DATA".L1_Press_0_24h := 0.0;
           "DATA".L1_Temp_0_2h := 0.0;
           "DATA".L1_Temp_2_4h := 0.0;
           "DATA".L1_Temp_4_6h := 0.0;
           "DATA".L1_Temp_6_8h := 0.0;
           "DATA".L1_Temp_8_10h := 0.0;
           "DATA".L1_Temp_10_12h := 0.0;
           "DATA".L1_Temp_12_14h := 0.0;
           "DATA".L1_Temp_14_16h := 0.0;
           "DATA".L1_Temp_16_18h := 0.0;
           "DATA".L1_Temp_18_20h := 0.0;
           "DATA".L1_Temp_20_22h := 0.0;
           "DATA".L1_Temp_22_24h := 0.0;
           "DATA".L1_Temp_0_24h := 0.0;
           "DATA".L1_Volume_0_2h := 0.0;
           "DATA".L1_Volume_2_4h := 0.0;
           "DATA".L1_Volume_4_6h := 0.0;
           "DATA".L1_Volume_6_8h := 0.0;
           "DATA".L1_Volume_8_10h := 0.0;
           "DATA".L1_Volume_10_12h := 0.0;
           "DATA".L1_Volume_12_14h := 0.0;
           "DATA".L1_Volume_14_16h := 0.0;
           "DATA".L1_Volume_16_18h := 0.0;
           "DATA".L1_Volume_18_20h := 0.0;
           "DATA".L1_Volume_20_22h := 0.0;
           "DATA".L1_Volume_22_24h := 0.0;
           "DATA".L1_Volume_0_24h := 0.0;
           "DATA".L1_Status_0_2h := 8;
           "DATA".L1_Status_2_4h := 8;
           "DATA".L1_Status_4_6h := 8;
           "DATA".L1_Status_6_8h := 8;
           "DATA".L1_Status_8_10h := 8;
           "DATA".L1_Status_10_12h := 8;
           "DATA".L1_Status_12_14h := 8;
           "DATA".L1_Status_14_16h := 8;
           "DATA".L1_Status_16_18h := 8;
           "DATA".L1_Status_18_20h := 8;
           "DATA".L1_Status_20_22h := 8;
           "DATA".L1_Status_22_24h := 8;
           "DATA".L1_Status_0_24h := 8;
           "DATA".L2_Volume_0_2h := 0.0;
           "DATA".L2_Volume_2_4h := 0.0;
           "DATA".L2_Volume_4_6h := 0.0;
           "DATA".L2_Volume_6_8h := 0.0;
           "DATA".L2_Volume_8_10h := 0.0;
           "DATA".L2_Volume_10_12h := 0.0;
           "DATA".L2_Volume_12_14h := 0.0;
           "DATA".L2_Volume_14_16h := 0.0;
           "DATA".L2_Volume_16_18h := 0.0;
           "DATA".L2_Volume_18_20h := 0.0;
           "DATA".L2_Volume_20_22h := 0.0;
           "DATA".L2_Volume_22_24h := 0.0;
           "DATA".L2_Volume_0_24h := 0.0;
           "DATA".L2_Status_0_2h := 8;
           "DATA".L2_Status_2_4h := 8;
           "DATA".L2_Status_4_6h := 8;
           "DATA".L2_Status_6_8h := 8;
           "DATA".L2_Status_8_10h := 8;
           "DATA".L2_Status_10_12h := 8;
           "DATA".L2_Status_12_14h := 8;
           "DATA".L2_Status_14_16h := 8;
           "DATA".L2_Status_16_18h := 8;
           "DATA".L2_Status_18_20h := 8;
           "DATA".L2_Status_20_22h := 8;
           "DATA".L2_Status_22_24h := 8;
           "DATA".L2_Status_0_24h := 8;
           "DATA".L3_Press_0_2h := 0.0;
           "DATA".L3_Press_2_4h := 0.0;
           "DATA".L3_Press_4_6h := 0.0;
           "DATA".L3_Press_6_8h := 0.0;
           "DATA".L3_Press_8_10h := 0.0;
           "DATA".L3_Press_10_12h := 0.0;
           "DATA".L3_Press_12_14h := 0.0;
           "DATA".L3_Press_14_16h := 0.0;
           "DATA".L3_Press_16_18h := 0.0;
           "DATA".L3_Press_18_20h := 0.0;
           "DATA".L3_Press_20_22h := 0.0;
           "DATA".L3_Press_22_24h := 0.0;
           "DATA".L3_Press_0_24h := 0.0;
           "DATA".L3_Temp_0_2h := 0.0;
           "DATA".L3_Temp_2_4h := 0.0;
           "DATA".L3_Temp_4_6h := 0.0;
           "DATA".L3_Temp_6_8h := 0.0;
           "DATA".L3_Temp_8_10h := 0.0;
           "DATA".L3_Temp_10_12h := 0.0;
           "DATA".L3_Temp_12_14h := 0.0;
           "DATA".L3_Temp_14_16h := 0.0;
           "DATA".L3_Temp_16_18h := 0.0;
           "DATA".L3_Temp_18_20h := 0.0;
           "DATA".L3_Temp_20_22h := 0.0;
           "DATA".L3_Temp_22_24h := 0.0;
           "DATA".L3_Temp_0_24h := 0.0;
           "DATA".L3_Volume_0_2h := 0.0;
           "DATA".L3_Volume_2_4h := 0.0;
           "DATA".L3_Volume_4_6h := 0.0;
           "DATA".L3_Volume_6_8h := 0.0;
           "DATA".L3_Volume_8_10h := 0.0;
           "DATA".L3_Volume_10_12h := 0.0;
           "DATA".L3_Volume_12_14h := 0.0;
           "DATA".L3_Volume_14_16h := 0.0;
           "DATA".L3_Volume_16_18h := 0.0;
           "DATA".L3_Volume_18_20h := 0.0;
           "DATA".L3_Volume_20_22h := 0.0;
           "DATA".L3_Volume_22_24h := 0.0;
           "DATA".L3_Volume_0_24h := 0.0;
           "DATA".L3_Status_0_2h := 8;
           "DATA".L3_Status_2_4h := 8;
           "DATA".L3_Status_4_6h := 8;
           "DATA".L3_Status_6_8h := 8;
           "DATA".L3_Status_8_10h := 8;
           "DATA".L3_Status_10_12h := 8;
           "DATA".L3_Status_12_14h := 8;
           "DATA".L3_Status_14_16h := 8;
           "DATA".L3_Status_16_18h := 8;
           "DATA".L3_Status_18_20h := 8;
           "DATA".L3_Status_20_22h := 8;
           "DATA".L3_Status_22_24h := 8;
           "DATA".L3_Status_0_24h := 8;



           "UVP_States".State := 61; // заходим в цикл чтения архива



         61:  // - запись параметров запроса на чтение архивных данных

               IF NOT "UVP_States".Client.Busy THEN
                   "UVP_States".ReqWriteCom.Mode := 1;
                   "UVP_States".ReqWriteCom.Data_ADDR := 47901;
                   "UVP_States".ReqWriteCom.Data_LEN := 14;
                   "ReqUVP" := 0;
                   "CopyWord"(NDBsrc := 13,
                              NDBdest := 14,
                              offset_src := 1000,
                              offset_dest := 52,
                              counter := 14);
                   "UVP_States".Answer := 0;
                   // Так как для УВП год вводится в формате "Число лет с 2000 г", а пользователю удобнее вводить полный год,
                   // принимаем год в обычном формате, а в УВП пишем число на 2000 меньше
                    "UVP_States".Data_PTR[4]  := "UVP_States".Data_PTR[4]  - 2000;
                    "UVP_States".Data_PTR[10] := "UVP_States".Data_PTR[10] - 2000;
                   "UVP_States".ClientMode := "UVP_States".ReqWriteCom;
                   "ReqUVP" := 1;
                   #NewState := 62;
               END_IF;

           62:  //  - ожидание записи параметров запроса на чтение архива в УВП, переход в режим записи формата запроса
               IF "UVP_States".Client.Done THEN
                   #NewState := 63;
                   //ELSIF #Request_Finished_with_Error THEN
                   //    #NewState := "UVP_States".ReqReadOpData_nextState;
               ELSE
                   ;
               END_IF;

           63: //  - запись формата запроса архивных данных (по нему стартует формирование архива в УВП)
               "UVP_States".ReqWriteCom.Mode := 1;
               "UVP_States".ReqWriteCom.Data_ADDR := 47915;
               "UVP_States".ReqWriteCom.Data_LEN := 1;
               "ReqUVP" := 0;
               "UVP_States".Data_PTR[0] := "UVP_States".Format;
               "UVP_States".ClientMode := "UVP_States".ReqWriteCom;
               "ReqUVP" := 1;
               // Можно начинать ждать архивных данных
               #NewState := 64;

           64: // - ожидание записи формата запроса       
               IF "UVP_States".Client.Done THEN
                   #NewState := 65;
               //ELSIF #Request_Finished_with_Error THEN
               //    #NewState := "UVP_States".ReqReadOpData_nextState;
               ELSE
                   ;
               END_IF;

           65: // чтение состояния готовности данных
               "UVP_States".ReqReadAns.Mode := 0;
               "UVP_States".ReqReadAns.Data_ADDR := 48001;
               "UVP_States".ReqReadAns.Data_LEN := 1;
               "ReqUVP" := 0;
               "UVP_States".ClientMode := "UVP_States".ReqReadAns;
               "ReqUVP" := 1;
               #NewState := 66;

           66: // обработка состояния готовности
               IF "UVP_States".Client.Done THEN
                   "UVP_States".Answer := "UVP_States".Data_PTR[0];
                   // Перекладываем статус запроса в DATA
                   IF ("UVP_Data".UVP1_Archives.UVP_line = 1) THEN
                       IF ("UVP_Data".UVP1_Archives.UVP_hour = 0) AND ("UVP_Data".UVP1_Archives.UVP_hour_end = 2) THEN
                           "DATA".L1_Status_0_2h := WORD_TO_INT("UVP_States".Answer);
                       ELSIF ("UVP_Data".UVP1_Archives.UVP_hour = 2) THEN
                           "DATA".L1_Status_2_4h := WORD_TO_INT("UVP_States".Answer);
                       ELSIF ("UVP_Data".UVP1_Archives.UVP_hour = 4) THEN
                           "DATA".L1_Status_4_6h := WORD_TO_INT("UVP_States".Answer);
                       ELSIF ("UVP_Data".UVP1_Archives.UVP_hour = 6) THEN
                           "DATA".L1_Status_6_8h := WORD_TO_INT("UVP_States".Answer);
                       ELSIF ("UVP_Data".UVP1_Archives.UVP_hour = 8) THEN
                           "DATA".L1_Status_8_10h := WORD_TO_INT("UVP_States".Answer);
                       ELSIF ("UVP_Data".UVP1_Archives.UVP_hour = 10) THEN
                           "DATA".L1_Status_10_12h := WORD_TO_INT("UVP_States".Answer);
                       ELSIF ("UVP_Data".UVP1_Archives.UVP_hour = 12) THEN
                           "DATA".L1_Status_12_14h := WORD_TO_INT("UVP_States".Answer);
                       ELSIF ("UVP_Data".UVP1_Archives.UVP_hour = 14) THEN
                           "DATA".L1_Status_14_16h := WORD_TO_INT("UVP_States".Answer);
                       ELSIF ("UVP_Data".UVP1_Archives.UVP_hour = 16) THEN
                           "DATA".L1_Status_16_18h := WORD_TO_INT("UVP_States".Answer);
                       ELSIF ("UVP_Data".UVP1_Archives.UVP_hour = 18) THEN
                           "DATA".L1_Status_18_20h := WORD_TO_INT("UVP_States".Answer);
                       ELSIF ("UVP_Data".UVP1_Archives.UVP_hour = 20) THEN
                           "DATA".L1_Status_20_22h := WORD_TO_INT("UVP_States".Answer);
                       ELSIF ("UVP_Data".UVP1_Archives.UVP_hour = 22) THEN
                           "DATA".L1_Status_22_24h := WORD_TO_INT("UVP_States".Answer);
                       ELSIF ("UVP_Data".UVP1_Archives.UVP_hour = 0) AND ("UVP_Data".UVP1_Archives.UVP_hour_end = 24) THEN
                           "DATA".L1_Status_0_24h := WORD_TO_INT("UVP_States".Answer);
                       END_IF;
                   ELSIF ("UVP_Data".UVP1_Archives.UVP_line = 2) THEN
                       IF ("UVP_Data".UVP1_Archives.UVP_hour = 0) AND ("UVP_Data".UVP1_Archives.UVP_hour_end = 2) THEN
                           "DATA".L2_Status_0_2h := WORD_TO_INT("UVP_States".Answer);
                       ELSIF ("UVP_Data".UVP1_Archives.UVP_hour = 2) THEN
                           "DATA".L2_Status_2_4h := WORD_TO_INT("UVP_States".Answer);
                       ELSIF ("UVP_Data".UVP1_Archives.UVP_hour = 4) THEN
                           "DATA".L2_Status_4_6h := WORD_TO_INT("UVP_States".Answer);
                       ELSIF ("UVP_Data".UVP1_Archives.UVP_hour = 6) THEN
                           "DATA".L2_Status_6_8h := WORD_TO_INT("UVP_States".Answer);
                       ELSIF ("UVP_Data".UVP1_Archives.UVP_hour = 8) THEN
                           "DATA".L2_Status_8_10h := WORD_TO_INT("UVP_States".Answer);
                       ELSIF ("UVP_Data".UVP1_Archives.UVP_hour = 10) THEN
                           "DATA".L2_Status_10_12h := WORD_TO_INT("UVP_States".Answer);
                       ELSIF ("UVP_Data".UVP1_Archives.UVP_hour = 12) THEN
                           "DATA".L2_Status_12_14h := WORD_TO_INT("UVP_States".Answer);
                       ELSIF ("UVP_Data".UVP1_Archives.UVP_hour = 14) THEN
                           "DATA".L2_Status_14_16h := WORD_TO_INT("UVP_States".Answer);
                       ELSIF ("UVP_Data".UVP1_Archives.UVP_hour = 16) THEN
                           "DATA".L2_Status_16_18h := WORD_TO_INT("UVP_States".Answer);
                       ELSIF ("UVP_Data".UVP1_Archives.UVP_hour = 18) THEN
                           "DATA".L2_Status_18_20h := WORD_TO_INT("UVP_States".Answer);
                       ELSIF ("UVP_Data".UVP1_Archives.UVP_hour = 20) THEN
                           "DATA".L2_Status_20_22h := WORD_TO_INT("UVP_States".Answer);
                       ELSIF ("UVP_Data".UVP1_Archives.UVP_hour = 22) THEN
                           "DATA".L2_Status_22_24h := WORD_TO_INT("UVP_States".Answer);
                       ELSIF ("UVP_Data".UVP1_Archives.UVP_hour = 0) AND ("UVP_Data".UVP1_Archives.UVP_hour_end = 24) THEN
                           "DATA".L2_Status_0_24h := WORD_TO_INT("UVP_States".Answer);
                       END_IF;
                   ELSIF ("UVP_Data".UVP1_Archives.UVP_line = 3) THEN
                       IF ("UVP_Data".UVP1_Archives.UVP_hour = 0) AND ("UVP_Data".UVP1_Archives.UVP_hour_end = 2) THEN
                           "DATA".L3_Status_0_2h := WORD_TO_INT("UVP_States".Answer);
                       ELSIF ("UVP_Data".UVP1_Archives.UVP_hour = 2) THEN
                           "DATA".L3_Status_2_4h := WORD_TO_INT("UVP_States".Answer);
                       ELSIF ("UVP_Data".UVP1_Archives.UVP_hour = 4) THEN
                           "DATA".L3_Status_4_6h := WORD_TO_INT("UVP_States".Answer);
                       ELSIF ("UVP_Data".UVP1_Archives.UVP_hour = 6) THEN
                           "DATA".L3_Status_6_8h := WORD_TO_INT("UVP_States".Answer);
                       ELSIF ("UVP_Data".UVP1_Archives.UVP_hour = 8) THEN
                           "DATA".L3_Status_8_10h := WORD_TO_INT("UVP_States".Answer);
                       ELSIF ("UVP_Data".UVP1_Archives.UVP_hour = 10) THEN
                           "DATA".L3_Status_10_12h := WORD_TO_INT("UVP_States".Answer);
                       ELSIF ("UVP_Data".UVP1_Archives.UVP_hour = 12) THEN
                           "DATA".L3_Status_12_14h := WORD_TO_INT("UVP_States".Answer);
                       ELSIF ("UVP_Data".UVP1_Archives.UVP_hour = 14) THEN
                           "DATA".L3_Status_14_16h := WORD_TO_INT("UVP_States".Answer);
                       ELSIF ("UVP_Data".UVP1_Archives.UVP_hour = 16) THEN
                           "DATA".L3_Status_16_18h := WORD_TO_INT("UVP_States".Answer);
                       ELSIF ("UVP_Data".UVP1_Archives.UVP_hour = 18) THEN
                           "DATA".L3_Status_18_20h := WORD_TO_INT("UVP_States".Answer);
                       ELSIF ("UVP_Data".UVP1_Archives.UVP_hour = 20) THEN
                           "DATA".L3_Status_20_22h := WORD_TO_INT("UVP_States".Answer);
                       ELSIF ("UVP_Data".UVP1_Archives.UVP_hour = 22) THEN
                           "DATA".L3_Status_22_24h := WORD_TO_INT("UVP_States".Answer);
                       ELSIF ("UVP_Data".UVP1_Archives.UVP_hour = 0) AND ("UVP_Data".UVP1_Archives.UVP_hour_end = 24) THEN
                           "DATA".L3_Status_0_24h := WORD_TO_INT("UVP_States".Answer);
                       END_IF;
                   END_IF;
                   IF "UVP_States".Answer = 16#0001 THEN         // идет сбор данных - читаем снова статус
                       #NewState := 65;
                   ELSE // данные готовы - переходим к их чтению
                       #NewState := 67;
                   END_IF;
               //ELSIF #Request_Finished_with_Error THEN
               //    #NewState := "UVP_States".ReqReadOpData_nextState;
               ELSE
                   ;
               END_IF;
         67: //  - запрашиваем строку архива
             IF NOT "UVP_States".Client.Busy THEN
               "UVP_States".ReqReadArcData.Mode := 0;
               "UVP_States".ReqReadArcData.Data_ADDR := 48003;
               "UVP_States".ReqReadArcData.Data_LEN := 120;
               "ReqUVP" := 0;
               "UVP_States".ClientMode := "UVP_States".ReqReadArcData;
               "ReqUVP" := 1;
               #NewState := 68;
             END_IF;

         68: // - обработка полученой строки архива
               IF "UVP_States".Client.Done THEN
                   "CopyWord"(NDBsrc := 14,
                              NDBdest := 14,
                              offset_src := 52,
                              offset_dest := 292,
                              counter := 120);

                   "len_String" := CHAR_TO_UINT("UVP_States".ArchArrayChar[1]) + (CHAR_TO_UINT("UVP_States".ArchArrayChar[0]) * 256) - 1;
                   #len := CHAR_TO_UINT("UVP_States".ArchArrayChar[1]) + (CHAR_TO_UINT("UVP_States".ArchArrayChar[0]) * 256) - 1;
                   Chars_TO_Strg(Chars := "UVP_States".ArchArrayChar,
                                 pChars := 2,
                                 Cnt := #len,
                                 Strg => "UVP_States".ArcDataString);
                   // данные кладём в нужную линию сразу
                   IF ("UVP_Data".UVP1_Archives.UVP_line = 1) THEN
                       "ParseString_2"(ClientIndex := 1);
                   ELSIF ("UVP_Data".UVP1_Archives.UVP_line = 2) THEN
                       ;
                       "ParseString_1"(ClientIndex := 2);
                   ELSIF ("UVP_Data".UVP1_Archives.UVP_line = 3) THEN
                       "ParseString_2"(ClientIndex := 3);
                   END_IF;
                   // Организуем цикл чтения архивов State 61-68, по окончании возвращаемся на циклическое чтение данных
                   IF NOT (("UVP_Data".UVP1_Archives.UVP_hour = 0) AND ("UVP_Data".UVP1_Archives.UVP_hour_end = 24) AND "UVP_Data".UVP1_Archives.UVP_line = 2) THEN
                       #NewState := 61;
                   ELSE
                       #NewState := 10;
                       "DATA".StartReadArchive := 0;
                   END_IF;

                   // Перекладываем данные в DATA
                   // ************* Линия 1 ********************************
                   IF ("UVP_Data".UVP1_Archives.UVP_line = 1) THEN
                       IF ("UVP_Data".UVP1_Archives.UVP_hour = 0) AND ("UVP_Data".UVP1_Archives.UVP_hour_end = 2) THEN
                           "DATA".L1_Press_0_2h := "UVP_States".ArhDataParsed[0, 0] / 1000000;
                           "DATA".L1_Temp_0_2h := "UVP_States".ArhDataParsed[0, 2];
                           "DATA".L1_Volume_0_2h := "UVP_States".ArhDataParsed[0, 4];
                           "UVP_Data".UVP1_Archives.UVP_hour := 2;
                           "UVP_Data".UVP1_Archives.UVP_hour_end := 4;
                       ELSIF ("UVP_Data".UVP1_Archives.UVP_hour = 2) THEN
                           "DATA".L1_Press_2_4h := "UVP_States".ArhDataParsed[0, 0] / 1000000;
                           "DATA".L1_Temp_2_4h := "UVP_States".ArhDataParsed[0, 2];
                           "DATA".L1_Volume_2_4h := "UVP_States".ArhDataParsed[0, 4];
                           "UVP_Data".UVP1_Archives.UVP_hour := 4;
                           "UVP_Data".UVP1_Archives.UVP_hour_end := 6;
                       ELSIF ("UVP_Data".UVP1_Archives.UVP_hour = 4) THEN
                           "DATA".L1_Press_4_6h := "UVP_States".ArhDataParsed[0, 0] / 1000000;
                           "DATA".L1_Temp_4_6h := "UVP_States".ArhDataParsed[0, 2];
                           "DATA".L1_Volume_4_6h := "UVP_States".ArhDataParsed[0, 4];
                           "UVP_Data".UVP1_Archives.UVP_hour := 6;
                           "UVP_Data".UVP1_Archives.UVP_hour_end := 8;
                       ELSIF ("UVP_Data".UVP1_Archives.UVP_hour = 6) THEN
                           "DATA".L1_Press_6_8h := "UVP_States".ArhDataParsed[0, 0] / 1000000;
                           "DATA".L1_Temp_6_8h := "UVP_States".ArhDataParsed[0, 2];
                           "DATA".L1_Volume_6_8h := "UVP_States".ArhDataParsed[0, 4];
                           "UVP_Data".UVP1_Archives.UVP_hour := 8;
                           "UVP_Data".UVP1_Archives.UVP_hour_end := 10;
                       ELSIF ("UVP_Data".UVP1_Archives.UVP_hour = 8) THEN
                           "DATA".L1_Press_8_10h := "UVP_States".ArhDataParsed[0, 0] / 1000000;
                           "DATA".L1_Temp_8_10h := "UVP_States".ArhDataParsed[0, 2];
                           "DATA".L1_Volume_8_10h := "UVP_States".ArhDataParsed[0, 4];
                           "UVP_Data".UVP1_Archives.UVP_hour := 10;
                           "UVP_Data".UVP1_Archives.UVP_hour_end := 12;
                       ELSIF ("UVP_Data".UVP1_Archives.UVP_hour = 10) THEN
                           "DATA".L1_Press_10_12h := "UVP_States".ArhDataParsed[0, 0] / 1000000;
                           "DATA".L1_Temp_10_12h := "UVP_States".ArhDataParsed[0, 2];
                           "DATA".L1_Volume_10_12h := "UVP_States".ArhDataParsed[0, 4];
                           "UVP_Data".UVP1_Archives.UVP_hour := 12;
                           "UVP_Data".UVP1_Archives.UVP_hour_end := 14;
                       ELSIF ("UVP_Data".UVP1_Archives.UVP_hour = 12) THEN
                           "DATA".L1_Press_12_14h := "UVP_States".ArhDataParsed[0, 0] / 1000000;
                           "DATA".L1_Temp_12_14h := "UVP_States".ArhDataParsed[0, 2];
                           "DATA".L1_Volume_12_14h := "UVP_States".ArhDataParsed[0, 4];
                           "UVP_Data".UVP1_Archives.UVP_hour := 14;
                           "UVP_Data".UVP1_Archives.UVP_hour_end := 16;
                       ELSIF ("UVP_Data".UVP1_Archives.UVP_hour = 14) THEN
                           "DATA".L1_Press_14_16h := "UVP_States".ArhDataParsed[0, 0] / 1000000;
                           "DATA".L1_Temp_14_16h := "UVP_States".ArhDataParsed[0, 2];
                           "DATA".L1_Volume_14_16h := "UVP_States".ArhDataParsed[0, 4];
                           "UVP_Data".UVP1_Archives.UVP_hour := 16;
                           "UVP_Data".UVP1_Archives.UVP_hour_end := 18;
                       ELSIF ("UVP_Data".UVP1_Archives.UVP_hour = 16) THEN
                           "DATA".L1_Press_16_18h := "UVP_States".ArhDataParsed[0, 0] / 1000000;
                           "DATA".L1_Temp_16_18h := "UVP_States".ArhDataParsed[0, 2];
                           "DATA".L1_Volume_16_18h := "UVP_States".ArhDataParsed[0, 4];
                           "UVP_Data".UVP1_Archives.UVP_hour := 18;
                           "UVP_Data".UVP1_Archives.UVP_hour_end := 20;
                       ELSIF ("UVP_Data".UVP1_Archives.UVP_hour = 18) THEN
                           "DATA".L1_Press_18_20h := "UVP_States".ArhDataParsed[0, 0] / 1000000;
                           "DATA".L1_Temp_18_20h := "UVP_States".ArhDataParsed[0, 2];
                           "DATA".L1_Volume_18_20h := "UVP_States".ArhDataParsed[0, 4];
                           "UVP_Data".UVP1_Archives.UVP_hour := 20;
                           "UVP_Data".UVP1_Archives.UVP_hour_end := 22;
                       ELSIF ("UVP_Data".UVP1_Archives.UVP_hour = 20) THEN
                           "DATA".L1_Press_20_22h := "UVP_States".ArhDataParsed[0, 0] / 1000000;
                           "DATA".L1_Temp_20_22h := "UVP_States".ArhDataParsed[0, 2];
                           "DATA".L1_Volume_20_22h := "UVP_States".ArhDataParsed[0, 4];
                           "UVP_Data".UVP1_Archives.UVP_hour := 22;
                           "UVP_Data".UVP1_Archives.UVP_hour_end := 24;
                       ELSIF ("UVP_Data".UVP1_Archives.UVP_hour = 22) THEN
                           "DATA".L1_Press_22_24h := "UVP_States".ArhDataParsed[0, 0] / 1000000;
                           "DATA".L1_Temp_22_24h := "UVP_States".ArhDataParsed[0, 2];
                           "DATA".L1_Volume_22_24h := "UVP_States".ArhDataParsed[0, 4];
                           "UVP_Data".UVP1_Archives.UVP_hour := 0;
                           "UVP_Data".UVP1_Archives.UVP_hour_end := 24;
                       ELSIF ("UVP_Data".UVP1_Archives.UVP_hour = 0) AND ("UVP_Data".UVP1_Archives.UVP_hour_end = 24) THEN
                           "DATA".L1_Press_0_24h := "UVP_States".ArhDataParsed[0, 0] / 1000000;
                           "DATA".L1_Temp_0_24h := "UVP_States".ArhDataParsed[0, 2];
                           "DATA".L1_Volume_0_24h := "UVP_States".ArhDataParsed[0, 4];
                           "UVP_Data".UVP1_Archives.UVP_hour := 0;
                           "UVP_Data".UVP1_Archives.UVP_hour_end := 2;
                           "UVP_Data".UVP1_Archives.UVP_line := 2;
                       END_IF;
                   // ************* Линия 2 *************************    
                   ELSIF ("UVP_Data".UVP1_Archives.UVP_line = 2) THEN
                       IF ("UVP_Data".UVP1_Archives.UVP_hour = 0) AND ("UVP_Data".UVP1_Archives.UVP_hour_end = 2) THEN
                           "DATA".L2_Volume_0_2h := "UVP_States".ArhDataParsed[1, 5];
                           "UVP_Data".UVP1_Archives.UVP_hour := 2;
                           "UVP_Data".UVP1_Archives.UVP_hour_end := 4;
                       ELSIF ("UVP_Data".UVP1_Archives.UVP_hour = 2) THEN
                           "DATA".L2_Volume_2_4h := "UVP_States".ArhDataParsed[1, 5];
                           "UVP_Data".UVP1_Archives.UVP_hour := 4;
                           "UVP_Data".UVP1_Archives.UVP_hour_end := 6;
                       ELSIF ("UVP_Data".UVP1_Archives.UVP_hour = 4) THEN
                           "DATA".L2_Volume_4_6h := "UVP_States".ArhDataParsed[1, 5];
                           "UVP_Data".UVP1_Archives.UVP_hour := 6;
                           "UVP_Data".UVP1_Archives.UVP_hour_end := 8;
                       ELSIF ("UVP_Data".UVP1_Archives.UVP_hour = 6) THEN
                           "DATA".L2_Volume_6_8h := "UVP_States".ArhDataParsed[1, 5];
                           "UVP_Data".UVP1_Archives.UVP_hour := 8;
                           "UVP_Data".UVP1_Archives.UVP_hour_end := 10;
                       ELSIF ("UVP_Data".UVP1_Archives.UVP_hour = 8) THEN
                           "DATA".L2_Volume_8_10h := "UVP_States".ArhDataParsed[1, 5];
                           "UVP_Data".UVP1_Archives.UVP_hour := 10;
                           "UVP_Data".UVP1_Archives.UVP_hour_end := 12;
                       ELSIF ("UVP_Data".UVP1_Archives.UVP_hour = 10) THEN
                           "DATA".L2_Volume_10_12h := "UVP_States".ArhDataParsed[1, 5];
                           "UVP_Data".UVP1_Archives.UVP_hour := 12;
                           "UVP_Data".UVP1_Archives.UVP_hour_end := 14;
                       ELSIF ("UVP_Data".UVP1_Archives.UVP_hour = 12) THEN
                           "DATA".L2_Volume_12_14h := "UVP_States".ArhDataParsed[1, 5];
                           "UVP_Data".UVP1_Archives.UVP_hour := 14;
                           "UVP_Data".UVP1_Archives.UVP_hour_end := 16;
                       ELSIF ("UVP_Data".UVP1_Archives.UVP_hour = 14) THEN
                           "DATA".L2_Volume_14_16h := "UVP_States".ArhDataParsed[1, 5];
                           "UVP_Data".UVP1_Archives.UVP_hour := 16;
                           "UVP_Data".UVP1_Archives.UVP_hour_end := 18;
                       ELSIF ("UVP_Data".UVP1_Archives.UVP_hour = 16) THEN
                           "DATA".L2_Volume_16_18h := "UVP_States".ArhDataParsed[1, 5];
                           "UVP_Data".UVP1_Archives.UVP_hour := 18;
                           "UVP_Data".UVP1_Archives.UVP_hour_end := 20;
                       ELSIF ("UVP_Data".UVP1_Archives.UVP_hour = 18) THEN
                           "DATA".L2_Volume_18_20h := "UVP_States".ArhDataParsed[1, 5];
                           "UVP_Data".UVP1_Archives.UVP_hour := 20;
                           "UVP_Data".UVP1_Archives.UVP_hour_end := 22;
                       ELSIF ("UVP_Data".UVP1_Archives.UVP_hour = 20) THEN
                           "DATA".L2_Volume_20_22h := "UVP_States".ArhDataParsed[1, 5];
                           "UVP_Data".UVP1_Archives.UVP_hour := 22;
                           "UVP_Data".UVP1_Archives.UVP_hour_end := 24;
                       ELSIF ("UVP_Data".UVP1_Archives.UVP_hour = 22) THEN
                           "DATA".L2_Volume_22_24h := "UVP_States".ArhDataParsed[1, 5];
                           "UVP_Data".UVP1_Archives.UVP_hour := 0;
                           "UVP_Data".UVP1_Archives.UVP_hour_end := 24;
                       ELSIF ("UVP_Data".UVP1_Archives.UVP_hour = 0) AND ("UVP_Data".UVP1_Archives.UVP_hour_end = 24) THEN
                           "DATA".L2_Volume_0_24h := "UVP_States".ArhDataParsed[1, 5];
                           "UVP_Data".UVP1_Archives.UVP_hour := 0;
                           "UVP_Data".UVP1_Archives.UVP_hour_end := 2;
                           "UVP_Data".UVP1_Archives.UVP_line := 3;
                       END_IF;
                       ;
                   // ************* Линия 3 ************************    
                   ELSIF ("UVP_Data".UVP1_Archives.UVP_line = 3) THEN
                       IF ("UVP_Data".UVP1_Archives.UVP_hour = 0) AND ("UVP_Data".UVP1_Archives.UVP_hour_end = 2) THEN
                           "DATA".L3_Press_0_2h := "UVP_States".ArhDataParsed[2, 0] / 1000000;
                           "DATA".L3_Temp_0_2h := "UVP_States".ArhDataParsed[2, 2];
                           "DATA".L3_Volume_0_2h := "UVP_States".ArhDataParsed[2, 4];
                           "UVP_Data".UVP1_Archives.UVP_hour := 2;
                           "UVP_Data".UVP1_Archives.UVP_hour_end := 4;
                       ELSIF ("UVP_Data".UVP1_Archives.UVP_hour = 2) THEN
                           "DATA".L3_Press_2_4h := "UVP_States".ArhDataParsed[2, 0] / 1000000;
                           "DATA".L3_Temp_2_4h := "UVP_States".ArhDataParsed[2, 2];
                           "DATA".L3_Volume_2_4h := "UVP_States".ArhDataParsed[2, 4];
                           "UVP_Data".UVP1_Archives.UVP_hour := 4;
                           "UVP_Data".UVP1_Archives.UVP_hour_end := 6;
                       ELSIF ("UVP_Data".UVP1_Archives.UVP_hour = 4) THEN
                           "DATA".L3_Press_4_6h := "UVP_States".ArhDataParsed[2, 0] / 1000000;
                           "DATA".L3_Temp_4_6h := "UVP_States".ArhDataParsed[2, 2];
                           "DATA".L3_Volume_4_6h := "UVP_States".ArhDataParsed[2, 4];
                           "UVP_Data".UVP1_Archives.UVP_hour := 6;
                           "UVP_Data".UVP1_Archives.UVP_hour_end := 8;
                       ELSIF ("UVP_Data".UVP1_Archives.UVP_hour = 6) THEN
                           "DATA".L3_Press_6_8h := "UVP_States".ArhDataParsed[2, 0] / 1000000;
                           "DATA".L3_Temp_6_8h := "UVP_States".ArhDataParsed[2, 2];
                           "DATA".L3_Volume_6_8h := "UVP_States".ArhDataParsed[2, 4];
                           "UVP_Data".UVP1_Archives.UVP_hour := 8;
                           "UVP_Data".UVP1_Archives.UVP_hour_end := 10;
                       ELSIF ("UVP_Data".UVP1_Archives.UVP_hour = 8) THEN
                           "DATA".L3_Press_8_10h := "UVP_States".ArhDataParsed[2, 0] / 1000000;
                           "DATA".L3_Temp_8_10h := "UVP_States".ArhDataParsed[2, 2];
                           "DATA".L3_Volume_8_10h := "UVP_States".ArhDataParsed[2, 4];
                           "UVP_Data".UVP1_Archives.UVP_hour := 10;
                           "UVP_Data".UVP1_Archives.UVP_hour_end := 12;
                       ELSIF ("UVP_Data".UVP1_Archives.UVP_hour = 10) THEN
                           "DATA".L3_Press_10_12h := "UVP_States".ArhDataParsed[2, 0] / 1000000;
                           "DATA".L3_Temp_10_12h := "UVP_States".ArhDataParsed[2, 2];
                           "DATA".L3_Volume_10_12h := "UVP_States".ArhDataParsed[2, 4];
                           "UVP_Data".UVP1_Archives.UVP_hour := 12;
                           "UVP_Data".UVP1_Archives.UVP_hour_end := 14;
                       ELSIF ("UVP_Data".UVP1_Archives.UVP_hour = 12) THEN
                           "DATA".L3_Press_12_14h := "UVP_States".ArhDataParsed[2, 0] / 1000000;
                           "DATA".L3_Temp_12_14h := "UVP_States".ArhDataParsed[2, 2];
                           "DATA".L3_Volume_12_14h := "UVP_States".ArhDataParsed[2, 4];
                           "UVP_Data".UVP1_Archives.UVP_hour := 14;
                           "UVP_Data".UVP1_Archives.UVP_hour_end := 16;
                       ELSIF ("UVP_Data".UVP1_Archives.UVP_hour = 14) THEN
                           "DATA".L3_Press_14_16h := "UVP_States".ArhDataParsed[2, 0] / 1000000;
                           "DATA".L3_Temp_14_16h := "UVP_States".ArhDataParsed[2, 2];
                           "DATA".L3_Volume_14_16h := "UVP_States".ArhDataParsed[2, 4];
                           "UVP_Data".UVP1_Archives.UVP_hour := 16;
                           "UVP_Data".UVP1_Archives.UVP_hour_end := 18;
                       ELSIF ("UVP_Data".UVP1_Archives.UVP_hour = 16) THEN
                           "DATA".L3_Press_16_18h := "UVP_States".ArhDataParsed[2, 0] / 1000000;
                           "DATA".L3_Temp_16_18h := "UVP_States".ArhDataParsed[2, 2];
                           "DATA".L3_Volume_16_18h := "UVP_States".ArhDataParsed[2, 4];
                           "UVP_Data".UVP1_Archives.UVP_hour := 18;
                           "UVP_Data".UVP1_Archives.UVP_hour_end := 20;
                       ELSIF ("UVP_Data".UVP1_Archives.UVP_hour = 18) THEN
                           "DATA".L3_Press_18_20h := "UVP_States".ArhDataParsed[2, 0] / 1000000;
                           "DATA".L3_Temp_18_20h := "UVP_States".ArhDataParsed[2, 2];
                           "DATA".L3_Volume_18_20h := "UVP_States".ArhDataParsed[2, 4];
                           "UVP_Data".UVP1_Archives.UVP_hour := 20;
                           "UVP_Data".UVP1_Archives.UVP_hour_end := 22;
                       ELSIF ("UVP_Data".UVP1_Archives.UVP_hour = 20) THEN
                           "DATA".L3_Press_20_22h := "UVP_States".ArhDataParsed[2, 0] / 1000000;
                           "DATA".L3_Temp_20_22h := "UVP_States".ArhDataParsed[2, 2];
                           "DATA".L3_Volume_20_22h := "UVP_States".ArhDataParsed[2, 4];
                           "UVP_Data".UVP1_Archives.UVP_hour := 22;
                           "UVP_Data".UVP1_Archives.UVP_hour_end := 24;
                       ELSIF ("UVP_Data".UVP1_Archives.UVP_hour = 22) THEN
                           "DATA".L3_Press_22_24h := "UVP_States".ArhDataParsed[2, 0] / 1000000;
                           "DATA".L3_Temp_22_24h := "UVP_States".ArhDataParsed[2, 2];
                           "DATA".L3_Volume_22_24h := "UVP_States".ArhDataParsed[2, 4];
                           "UVP_Data".UVP1_Archives.UVP_hour := 0;
                           "UVP_Data".UVP1_Archives.UVP_hour_end := 24;
                       ELSIF ("UVP_Data".UVP1_Archives.UVP_hour = 0) AND ("UVP_Data".UVP1_Archives.UVP_hour_end = 24) THEN
                           "DATA".L3_Press_0_24h := "UVP_States".ArhDataParsed[2, 0] / 1000000;
                           "DATA".L3_Temp_0_24h := "UVP_States".ArhDataParsed[2, 2];
                           "DATA".L3_Volume_0_24h := "UVP_States".ArhDataParsed[2, 4];
                           "UVP_Data".UVP1_Archives.UVP_hour := 0;
                           "UVP_Data".UVP1_Archives.UVP_hour_end := 2;
                           "UVP_Data".UVP1_Archives.UVP_line := 1;
                       END_IF;
                   END_IF;



                   //#NewState := "UVP_States".ReqReadOpData_nextState;

               //ELSIF #Request_Finished_with_Error THEN
                   //#NewState := "UVP_States".ReqReadOpData_nextState;
               ELSE
                   ;
               END_IF;

    // Если случайно State кривой - начнём с начала
   ELSE
       ;
       #NewState := 10;
   END_CASE;

   "PrevState" := "UVP_States".State;

   IF #NewState >= 0 THEN
       "UVP_States".State := #NewState;
   END_IF;

   ////////
   (*"UVP_States".ArcDataStOp := "UVP_States".ArcDataString;
   "len2" := LEN("UVP_States".ArcDataString);
   "Point_test" :=FIND(IN1 := "UVP_States".ArcDataString, IN2 := ';');
   "UVP_States".SubString[1] := LEFT(IN := "UVP_States".ArcDataString, L := "Point_test" - 1);
   IF NOT "Test_bit" THEN
       "UVP_States".ArcDataString := DELETE(IN := "UVP_States".ArcDataString, L := "Point_test", P := 1);
       "Test_bit" := true;
   END_IF;*)

   (*"len2" := LEN("UVP_States".ArcDataString);
   //WHILE ("Test_int" < 3) OR (LEN("UVP_States".ArcDataString) > 0) DO
   WHILE ("Test_int" < 7) DO
       "Point_test" := FIND(IN1 := "UVP_States".ArcDataString, IN2 := ';');
       //IF ("Point_test" = 0) THEN
           //"UVP_States".SubString["Test_int"] := LEFT(IN := "UVP_States".ArcDataString, L := LEN("UVP_States".ArcDataString));
           //"UVP_States".ArcDataString := DELETE(IN := "UVP_States".ArcDataString, L := LEN("UVP_States".ArcDataString), P := 1);
       //ELSE
           "UVP_States".SubString["Test_int"] := LEFT(IN := "UVP_States".ArcDataString, L := "Point_test" - 1);
           "UVP_States".ArcDataString := DELETE(IN := "UVP_States".ArcDataString, L := "Point_test", P := 1);
       //END_IF;
       "Test_int" := "Test_int" + 1;
   END_WHILE;*)
END_FUNCTION

FUNCTION "REG_Processing" : Void   // FC10, SCL
{ S7_Optimized_Access := 'FALSE' }
VERSION : 0.1
   VAR_TEMP
      Request_Finished : Bool;
      Request_Finished_with_Error : Bool;
   END_VAR
BEGIN
   // Если порт не поднят, поднимаем
   IF NOT "Modbus_Comm_Load_Regs".DONE THEN
       "Modbus_Comm_Load_Regs".MODE := 4; // Operating mode 4 = Half duplex (RS485) two-wire mode
       "Modbus_Comm_Load_Regs"(REQ := true,
                               "PORT" := "PortSettings".Regs."Port",
                               BAUD := "PortSettings".Regs.Baud,
                               PARITY := "PortSettings".Regs.Parity,
                               FLOW_CTRL := 0,
                               RTS_ON_DLY := 0,
                               RTS_OFF_DLY := 0,
                               RESP_TO := 1000,
                               DONE => "PortSettings".Regs.Done,
                               ERROR => "PortSettings".Regs.Error,
                               STATUS => "PortSettings".Regs.Status,
                               MB_DB := "Modbus_Master_Regs".MB_DB);
   END_IF;

   // *********************************************Диагностика ошибок**********************************************************
   #Request_Finished := "REG_Master".Settings.Done OR "REG_Master".Settings.Error;
   // признак завершения цикла работы чтения/записи с ошибкой
   #Request_Finished_with_Error :=
   "REG_Master".Settings.Error AND ((("REG_Master".Settings.Status = 16#8380)) OR (("REG_Master".Settings.Status = 16#8381)) OR (("REG_Master".Settings.Status = 16#8382)) OR (("REG_Master".Settings.Status = 16#8383)) OR (("REG_Master".Settings.Status = 16#8384)) OR (("REG_Master".Settings.Status = 16#8385)) OR (("REG_Master".Settings.Status = 16#8386)) OR (("REG_Master".Settings.Status = 16#8387)) OR (("REG_Master".Settings.Status = 16#8388)));

   // блок обработки ошибки связи
   IF (("REG_Master".Settings.Status <> 16#0000) AND ("REG_Master".Settings.Status <> 16#7000) AND ("REG_Master".Settings.Status <> 16#7001) AND ("REG_Master".Settings.Status <> 16#7002)) THEN
       IF "REG_Master".Settings.MB_Addr = 1 THEN
           "REG_Master".PCV300_error := TRUE;
       END_IF;
       IF "REG_Master".Settings.MB_Addr = 2 THEN
           "REG_Master".LCV300_error := TRUE;
       END_IF;
   END_IF;

   // блок сброса ошибки связи
   IF "REG_Master".Settings.Done AND (NOT "REG_Master".Settings.Error) THEN
       IF "REG_Master".Settings.MB_Addr = 1 THEN
           "REG_Master".PCV300_error := false;
       END_IF;
       IF "REG_Master".Settings.MB_Addr = 2 THEN
           "REG_Master".LCV300_error := false;
       END_IF;
   END_IF;

   //*********************************************************************************************

   // 10 - чтение с регулятора PCV300, сетевой адрес 1
   // 11 - чтение с регулятора LCV300, сетевой адрес 2 
   // 13 - запись в PCV300 задания положения
   // 14 - запись в LCV300 задания положения 

   IF "REG_Master".State = 10 THEN

       IF "REG_Master".State = 10 AND "REG_Master".reg_PCV300_err = true THEN
           IF "REG_Master".count_PCV300 < 1000 THEN
               "REG_Master".State := 11;
               "REG_Master".count_PCV300 := "REG_Master".count_PCV300 + 1;
           ELSIF "REG_Master".count_PCV300 >= 1000 THEN
               "REG_Master".count_PCV300 := 0;
               "REG_Master".reg_PCV300_err := false;
           END_IF;
       END_IF;

       IF "REG_Master".State = 10 AND "REG_Master".reg_PCV300_err = false THEN
           "REG_Master".MasterMode.Mode := 0;
           "REG_Master".Settings.MB_Addr := 1;
           "REG_Master".MasterMode.Data_Addr := 31001;
           "REG_Master".MasterMode.Data_Len := 3;
           "REG_Master".Data_offset := 2;
           "REG_Master".Register := 3;
           "REG_Master".Next_State := 11;
           "REG_Master".reqREGmaster := 1;
       END_IF;
   END_IF;

   IF "REG_Master".State = 11 THEN
       IF "REG_Master".State = 11 AND "REG_Master".reg_LCV300_err = true THEN
           IF "REG_Master".count_LCV300 < 1000 THEN
               "REG_Master".State := 13;
               "REG_Master".count_LCV300 := "REG_Master".count_LCV300 + 1;
           ELSIF "REG_Master".count_LCV300 >= 1000 THEN
               "REG_Master".count_LCV300 := 0;
               "REG_Master".reg_LCV300_err := false;
           END_IF;
       END_IF;

       IF "REG_Master".State = 11 AND "REG_Master".reg_LCV300_err = false THEN
           "REG_Master".MasterMode.Mode := 0;
           "REG_Master".Settings.MB_Addr := 2;
           "REG_Master".MasterMode.Data_Addr := 31001;
           "REG_Master".MasterMode.Data_Len := 3;
           "REG_Master".Data_offset := 14;
           "REG_Master".Register := 3;
           "REG_Master".Next_State := 13;
           "REG_Master".reqREGmaster := 1;
       END_IF;
   END_IF;

   IF "REG_Master".State = 13 THEN
       // переходим на запись положений (SP)

       IF "REG_Master".State = 13 AND "REG_Master".reg_PCV300_err = true THEN
           "REG_Master".State := 14;
       END_IF;

       IF "REG_Master".State = 13 AND "REG_Master".reg_PCV300_err = false THEN
           "REG_Master".MasterMode.Mode := 1;
           "REG_Master".Settings.MB_Addr := 1;
           "REG_Master".MasterMode.Data_Addr := 41001;
           "REG_Master".MasterMode.Data_Len := 2;
           "REG_Master".Register := 1;
           "REG_Master".Next_State := 14;
           %DB16.DBW6 := 1024;
           "CopyWord"(NDBsrc := 15,
                      NDBdest := 16,
                      offset_src := 12,
                      offset_dest := 8,
                      counter := "REG_Master".Register);
           "REG_Master".reqREGmaster := 1;
       END_IF;
   END_IF;

   IF "REG_Master".State = 14 THEN
       IF "REG_Master".State = 14 AND "REG_Master".reg_LCV300_err = true THEN
           "REG_Master".State := 10;
       END_IF;

       IF "REG_Master".State = 14 AND "REG_Master".reg_LCV300_err = false THEN
           "REG_Master".MasterMode.Mode := 1;
           "REG_Master".Settings.MB_Addr := 2;
           "REG_Master".MasterMode.Data_Addr := 41001;
           "REG_Master".MasterMode.Data_Len := 2;
           "REG_Master".Register := 1;
           "REG_Master".Next_State := 10;
           %DB16.DBW6 := 1024;
           "CopyWord"(NDBsrc := 15,
                      NDBdest := 16,
                      offset_src := 24,
                      offset_dest := 8,
                      counter := "REG_Master".Register);
           "REG_Master".reqREGmaster := 1;
       END_IF;
   END_IF;

   IF "REG_Master".State = 10 OR "REG_Master".State = 11 OR "REG_Master".State = 12 THEN

       // обработка принятых данных
       IF "REG_Master".Settings.Done THEN
           IF "REG_Master".reg_PCV300_err = false OR "REG_Master".reg_LCV300_err = false THEN
               //"SwapWord"(NDB := 57,
               //           offset := 6,
               //           counter := 1);
               //"SwapWord"(NDB := 57,
               //           offset := 10,
               //           counter := 1);
               "CopyWord"(NDBsrc := 16,//пересылка из буфера в DBшку
                          NDBdest := 15,
                          offset_src := 6,
                          offset_dest := "REG_Master".Data_offset,
                          counter := "REG_Master".Register);

               IF ("REG_Master".State = 10) THEN
                   "REG_Master".PCV300_done_count := "REG_Master".PCV300_done_count + 1;
                   "REG_Master".PCV300_error := false;
                   IF ("REG_Master".PCV300_done_count >= 10000) THEN
                       "REG_Master".PCV300_done_count := 0;
                   END_IF;
               ELSIF ("REG_Master".State = 11) THEN
                   "REG_Master".LCV300_done_count := "REG_Master".LCV300_done_count + 1;
                   "REG_Master".LCV300_error := false;
                   IF ("REG_Master".LCV300_done_count >= 10000) THEN
                       "REG_Master".LCV300_done_count := 0;
                   END_IF;
               END_IF;

               IF NOT "REG_Master".Settings.Busy THEN
                   "REG_Master".State := "REG_Master".Next_State;
                   "REG_Master".reqREGmaster := 0;
               END_IF;
           ELSIF #Request_Finished_with_Error THEN
               "REG_Master".State := "REG_Master".Next_State;
               "REG_Master".reqREGmaster := 0;
           END_IF;
       END_IF;

       IF "REG_Master".State = 10 OR "REG_Master".State = 11 OR "REG_Master".State = 12 THEN
           IF ("REG_Master".Settings.Busy OR "REG_Master".Settings.Error) THEN
               "Timer_Busy_Modbus_Reg".TON(IN := true, PT := t#5s);
               IF "Timer_Busy_Modbus_Reg".Q THEN

                   IF "REG_Master".State = 10 THEN
                       "REG_Master".reg_PCV300_err := true;
                       "REG_Master".count_PCV300 := 0;
                       "REG_Master".PCV300_error := true;
                   END_IF;

                   IF "REG_Master".State = 11 THEN
                       "REG_Master".reg_LCV300_err := true;
                       "REG_Master".count_LCV300 := 0;
                       "REG_Master".LCV300_error := true;
                   END_IF;

                   "REG_Master".reqREGmaster := 0;
                   "REG_Master".State := "REG_Master".Next_State;
                   "Timer_Busy_Modbus_Reg".TON(IN := false, PT := t#5s);
               END_IF;
           ELSE
               "Timer_Busy_Modbus_Reg".TON(IN := false, PT := t#5s);
           END_IF;
       END_IF;

   END_IF;


   IF "REG_Master".State = 13 OR "REG_Master".State = 14 OR "REG_Master".State = 15 THEN

       //"REG_Master".MasterMode.Mode := 1;

       IF "REG_Master".Settings.Done THEN
           IF "REG_Master".State = 13 OR "REG_Master".State = 14 OR "REG_Master".State = 15 THEN
               IF NOT "REG_Master".Settings.Busy THEN
                   "REG_Master".State := "REG_Master".Next_State;
                   "REG_Master".reqREGmaster := 0;
               ELSIF #Request_Finished_with_Error THEN
                   "REG_Master".State := "REG_Master".Next_State;
                   "REG_Master".reqREGmaster := 0;
               END_IF;
           END_IF;
       END_IF;

       IF ("REG_Master".Settings.Busy OR "REG_Master".Settings.Error) THEN
           "Timer_Busy_Modbus_Reg2".TON(IN := true, PT := t#5s);
           IF "Timer_Busy_Modbus_Reg2".Q THEN

               //-----На случай если данные прочитались с регулятора, но не записались--------------
               IF "REG_Master".State = 13 THEN
                   "REG_Master".reg_PCV300_err := true;
                   "REG_Master".count_PCV300 := 0;
                   "REG_Master".PCV300_error := true;
               END_IF;

               IF "REG_Master".State = 14 THEN
                   "REG_Master".reg_LCV300_err := true;
                   "REG_Master".count_LCV300 := 0;
                   "REG_Master".LCV300_error := true;
               END_IF;

               //----------------------------------------------------------------------------------

               "REG_Master".reqREGmaster := 0;
               "REG_Master".State := "REG_Master".Next_State;
               "Timer_Busy_Modbus_Reg2".TON(IN := false, PT := t#5s);
           END_IF;
       ELSE
           "Timer_Busy_Modbus_Reg2".TON(IN := false, PT := t#5s);
       END_IF;
   END_IF;


   // приведение положения регулятора с 100% шкале

   "REG_Data".PCV300_Pologenie_ok := INT_TO_REAL("REG_Data".PCV300_Pologenie) / 10;
   "REG_Data".LCV300_Pologenie_ok := INT_TO_REAL("REG_Data".LCV300_Pologenie) / 10;
   //
   IF "REG_Data".PCV300_Pologenie_ok > 98.5 THEN
       "REG_Data".PCV300_Pologenie_ok := 100.0;
   END_IF;
   IF "REG_Data".LCV300_Pologenie_ok > 98.5 THEN
       "REG_Data".LCV300_Pologenie_ok := 100.0;
   END_IF;


